C09108=1053.623,-71.148,432.234,170.544,29.693,155.607
C09109=1053.617,-71.397,432.246,170.542,29.692,155.607
C09110=1053.611,-71.647,432.257,170.540,29.691,155.607
C09111=1053.606,-71.896,432.269,170.538,29.689,155.606
C09112=1053.599,-72.147,432.280,170.536,29.688,155.606
C09113=1053.593,-72.396,432.292,170.535,29.686,155.606
C09114=1053.587,-72.646,432.303,170.533,29.685,155.606
C09115=1053.582,-72.895,432.315,170.531,29.684,155.606
C09116=1053.575,-73.145,432.327,170.529,29.683,155.606
C09117=1053.569,-73.394,432.338,170.527,29.681,155.606
C09118=1053.563,-73.644,432.349,170.524,29.679,155.606
C09119=1053.556,-73.894,432.361,170.523,29.679,155.606
C09120=1053.551,-74.144,432.373,170.521,29.677,155.606
C09121=1053.545,-74.394,432.384,170.519,29.676,155.606
C09122=1053.538,-74.643,432.394,170.517,29.675,155.605
C09123=1053.532,-74.892,432.406,170.515,29.673,155.605
C09124=1053.526,-75.142,432.417,170.513,29.672,155.605
C09125=1053.519,-75.392,432.429,170.511,29.671,155.605
C09126=1053.514,-75.641,432.440,170.510,29.670,155.605
C09127=1053.507,-75.891,432.451,170.508,29.669,155.605
C09128=1053.501,-76.141,432.462,170.505,29.668,155.605
C09129=1053.495,-76.390,432.474,170.503,29.666,155.605
C09130=1053.489,-76.640,432.485,170.501,29.665,155.605
C09131=1053.483,-76.890,432.496,170.499,29.663,155.605
C09132=1053.476,-77.140,432.508,170.498,29.662,155.605
C09133=1053.470,-77.389,432.519,170.496,29.661,155.605
C09134=1053.464,-77.639,432.530,170.494,29.660,155.604
C09135=1053.458,-77.889,432.541,170.492,29.659,155.604
C09136=1053.452,-78.138,432.553,170.490,29.658,155.604
C09137=1053.446,-78.388,432.564,170.487,29.657,155.604
C09138=1053.440,-78.638,432.575,170.486,29.655,155.604
C09139=1053.434,-78.887,432.586,170.484,29.654,155.604
C09140=1053.427,-79.137,432.598,170.482,29.653,155.604
C09141=1053.421,-79.386,432.609,170.480,29.651,155.604
C09142=1053.415,-79.637,432.620,170.478,29.651,155.604
C09143=1053.409,-79.886,432.631,170.476,29.650,155.604
C09144=1053.402,-80.136,432.642,170.474,29.649,155.604
C09145=1053.396,-80.385,432.653,170.473,29.647,155.604
C09146=1053.390,-80.635,432.665,170.470,29.646,155.604
C09147=1053.384,-80.885,432.675,170.468,29.645,155.604
C09148=1053.377,-81.134,432.686,170.466,29.644,155.604
C09149=1053.371,-81.384,432.697,170.464,29.643,155.604
C09150=1053.365,-81.634,432.708,170.462,29.642,155.604
C09151=1053.359,-81.884,432.719,170.460,29.641,155.604
C09152=1053.352,-82.134,432.730,170.459,29.640,155.604
C09153=1053.346,-82.382,432.741,170.457,29.638,155.603
C09154=1053.339,-82.666,432.754,170.454,29.637,155.603
C09155=1053.332,-82.949,432.766,170.452,29.636,155.603
C09156=1053.325,-83.233,432.778,170.449,29.635,155.603
C09157=1053.318,-83.517,432.791,170.447,29.633,155.603
C09158=1053.312,-83.767,432.802,170.446,29.632,155.603
C09159=1053.305,-84.017,432.812,170.444,29.631,155.603
C09160=1053.299,-84.266,432.823,170.441,29.630,155.603
C09161=1053.293,-84.516,432.835,170.439,29.629,155.603
C09162=1053.286,-84.766,432.845,170.437,29.628,155.603
C09163=1053.281,-85.015,432.856,170.435,29.627,155.603
C09164=1053.274,-85.265,432.867,170.433,29.626,155.603
C09165=1053.268,-85.515,432.877,170.431,29.625,155.603
C09166=1053.262,-85.765,432.889,170.430,29.624,155.603
C09167=1053.256,-86.014,432.899,170.428,29.623,155.603
C09168=1053.250,-86.264,432.910,170.425,29.622,155.603
C09169=1053.243,-86.514,432.921,170.423,29.621,155.603
C09170=1053.237,-86.763,432.932,170.421,29.620,155.603
C09171=1053.231,-87.013,432.943,170.419,29.619,155.603
C09172=1053.224,-87.262,432.953,170.417,29.618,155.603
C09173=1053.219,-87.512,432.964,170.416,29.617,155.603
C09174=1053.212,-87.762,432.975,170.414,29.616,155.603
C09175=1053.206,-88.011,432.986,170.411,29.615,155.603
C09176=1053.200,-88.261,432.997,170.409,29.614,155.603
C09177=1053.194,-88.512,433.007,170.407,29.613,155.602
C09178=1053.188,-88.761,433.017,170.405,29.612,155.602
C09179=1053.182,-89.010,433.028,170.403,29.611,155.602
C09180=1053.176,-89.260,433.040,170.402,29.610,155.602
C09181=1053.169,-89.510,433.050,170.400,29.609,155.602
C09182=1053.163,-89.759,433.061,170.397,29.608,155.602
C09183=1053.156,-90.009,433.071,170.395,29.607,155.602
C09184=1053.151,-90.258,433.082,170.393,29.606,155.602
C09185=1053.145,-90.509,433.092,170.391,29.605,155.602
C09186=1053.138,-90.758,433.103,170.389,29.604,155.602
C09187=1053.132,-91.008,433.114,170.388,29.603,155.602
C09188=1053.127,-91.257,433.125,170.386,29.602,155.602
C09189=1053.119,-91.507,433.135,170.384,29.601,155.602
C09190=1053.114,-91.757,433.146,170.381,29.600,155.602
C09191=1053.108,-92.007,433.156,170.379,29.599,155.602
C09192=1053.102,-92.256,433.167,170.377,29.598,155.602
C09193=1053.095,-92.506,433.178,170.375,29.597,155.602
C09194=1053.089,-92.755,433.188,170.374,29.596,155.602
C09195=1053.084,-93.006,433.198,170.372,29.595,155.602
C09196=1053.078,-93.255,433.209,170.370,29.594,155.602
C09197=1053.071,-93.505,433.220,170.367,29.593,155.602
C09198=1053.065,-93.754,433.231,170.365,29.592,155.602
C09199=1053.059,-94.004,433.240,170.363,29.591,155.602
C09200=1053.053,-94.254,433.251,170.361,29.590,155.602
C09201=1053.047,-94.504,433.263,170.359,29.589,155.602
C09202=1053.041,-94.754,433.272,170.358,29.588,155.602
C09203=1053.035,-95.003,433.283,170.355,29.587,155.602
C09204=1053.028,-95.252,433.293,170.353,29.586,155.602
C09205=1053.023,-95.503,433.303,170.351,29.586,155.602
C09206=1053.017,-95.753,433.315,170.349,29.585,155.602
C09207=1053.010,-96.002,433.325,170.347,29.584,155.602
C09208=1053.004,-96.251,433.336,170.345,29.583,155.602
C09209=1052.998,-96.501,433.345,170.344,29.582,155.602
C09210=1052.992,-96.751,433.356,170.341,29.580,155.602
C09211=1052.986,-97.001,433.367,170.339,29.579,155.602
C09212=1052.980,-97.251,433.377,170.337,29.579,155.602
C09213=1052.974,-97.500,433.388,170.335,29.578,155.602
C09214=1052.968,-97.750,433.398,170.333,29.577,155.602
C09215=1052.962,-97.999,433.408,170.331,29.576,155.602
C09216=1052.956,-98.250,433.418,170.329,29.576,155.602
C09217=1052.949,-98.499,433.429,170.327,29.574,155.602
C09218=1052.942,-98.785,433.440,170.325,29.573,155.602
C09219=1052.935,-99.071,433.452,170.322,29.573,155.602
C09220=1052.928,-99.357,433.463,170.320,29.572,155.602
C09221=1052.921,-99.643,433.475,170.317,29.571,155.602
C09222=1052.915,-99.893,433.486,170.315,29.570,155.602
C09223=1052.909,-100.142,433.496,170.313,29.569,155.602
C09224=1052.902,-100.392,433.506,170.311,29.568,155.602
C09225=1052.896,-100.642,433.517,170.310,29.568,155.602
C09226=1052.890,-100.891,433.527,170.308,29.567,155.602
C09227=1052.884,-101.141,433.537,170.305,29.566,155.602
C09228=1052.878,-101.391,433.547,170.303,29.565,155.602
C09229=1052.872,-101.641,433.557,170.301,29.564,155.602
C09230=1052.865,-101.890,433.567,170.299,29.564,155.602
C09231=1052.860,-102.141,433.577,170.297,29.563,155.602
C09232=1052.853,-102.390,433.588,170.295,29.562,155.602
C09233=1052.847,-102.640,433.597,170.293,29.561,155.602
C09234=1052.841,-102.889,433.608,170.291,29.560,155.602
C09235=1052.835,-103.139,433.618,170.289,29.560,155.602
C09236=1052.828,-103.388,433.628,170.287,29.559,155.602
C09237=1052.823,-103.638,433.638,170.285,29.559,155.602
C09238=1052.817,-103.888,433.648,170.283,29.558,155.602
C09239=1052.810,-104.138,433.658,170.280,29.556,155.602
C09240=1052.804,-104.388,433.668,170.278,29.556,155.602
C09241=1052.798,-104.638,433.678,170.276,29.555,155.602
C09242=1052.792,-104.887,433.688,170.275,29.555,155.602
C09243=1052.786,-105.137,433.698,170.273,29.554,155.602
C09244=1052.780,-105.386,433.709,170.271,29.553,155.602
C09245=1052.774,-105.636,433.718,170.268,29.552,155.602
C09246=1052.767,-105.886,433.728,170.266,29.552,155.602
C09247=1052.761,-106.135,433.738,170.264,29.551,155.602
C09248=1052.756,-106.385,433.748,170.262,29.550,155.602
C09249=1052.749,-106.635,433.758,170.260,29.549,155.602
C09250=1052.743,-106.885,433.767,170.258,29.549,155.602
C09251=1052.737,-107.134,433.778,170.256,29.548,155.602
C09252=1052.731,-107.384,433.788,170.254,29.547,155.602
C09253=1052.725,-107.634,433.798,170.252,29.547,155.602
C09254=1052.718,-107.884,433.808,170.250,29.546,155.602
C09255=1052.712,-108.133,433.818,170.248,29.546,155.602
C09256=1052.706,-108.383,433.827,170.245,29.544,155.602
C09257=1052.700,-108.633,433.837,170.243,29.544,155.603
C09258=1052.693,-108.883,433.846,170.241,29.544,155.603
C09259=1052.687,-109.132,433.857,170.239,29.543,155.603
C09260=1052.681,-109.382,433.867,170.237,29.542,155.603
C09261=1052.675,-109.632,433.876,170.236,29.542,155.603
C09262=1052.669,-109.882,433.886,170.233,29.541,155.603
C09263=1052.663,-110.131,433.896,170.231,29.540,155.603
C09264=1052.656,-110.381,433.906,170.229,29.540,155.603
C09265=1052.650,-110.630,433.915,170.227,29.539,155.603
C09266=1052.644,-110.880,433.925,170.225,29.539,155.603
C09267=1052.638,-111.130,433.935,170.222,29.538,155.603
C09268=1052.632,-111.380,433.944,170.220,29.538,155.603
C09269=1052.626,-111.630,433.954,170.218,29.537,155.603
C09270=1052.620,-111.879,433.965,170.217,29.536,155.603
C09271=1052.614,-112.129,433.974,170.215,29.536,155.603
C09272=1052.607,-112.379,433.984,170.213,29.535,155.603
C09273=1052.601,-112.629,433.993,170.210,29.534,155.603
C09274=1052.595,-112.878,434.003,170.208,29.534,155.603
C09275=1052.589,-113.128,434.012,170.206,29.534,155.603
C09276=1052.583,-113.378,434.022,170.204,29.533,155.603
C09277=1052.577,-113.628,434.032,170.202,29.532,155.603
C09278=1052.570,-113.878,434.041,170.199,29.532,155.604
C09279=1052.564,-114.127,434.051,170.197,29.531,155.604
C09280=1052.558,-114.377,434.060,170.196,29.530,155.604
C09281=1052.552,-114.626,434.070,170.194,29.530,155.604
C09282=1052.545,-114.911,434.081,170.191,29.529,155.604
C09283=1052.538,-115.194,434.092,170.189,29.529,155.604
C09284=1052.531,-115.478,434.103,170.186,29.528,155.604
C09285=1052.524,-115.763,434.113,170.184,29.527,155.604
C09286=1052.518,-116.013,434.123,170.182,29.527,155.604
C09287=1052.512,-116.262,434.132,170.180,29.527,155.604
C09288=1052.506,-116.511,434.142,170.177,29.526,155.604
C09289=1052.500,-116.761,434.151,170.175,29.526,155.604
C09290=1052.494,-117.011,434.161,170.173,29.525,155.604
C09291=1052.488,-117.261,434.170,170.172,29.525,155.604
C09292=1052.482,-117.511,434.180,170.170,29.524,155.605
C09293=1052.475,-117.760,434.189,170.167,29.523,155.605
C09294=1052.469,-118.010,434.199,170.165,29.523,155.605
C09295=1052.463,-118.260,434.209,170.163,29.522,155.605
C09296=1052.457,-118.510,434.218,170.161,29.522,155.605
C09297=1052.450,-118.759,434.227,170.159,29.522,155.605
C09298=1052.444,-119.008,434.236,170.156,29.521,155.605
C09299=1052.438,-119.258,434.246,170.154,29.521,155.605
C09300=1052.432,-119.509,434.255,170.152,29.520,155.605
C09301=1052.426,-119.758,434.264,170.150,29.520,155.605
C09302=1052.420,-120.008,434.274,170.149,29.520,155.605
C09303=1052.414,-120.258,434.283,170.146,29.519,155.605
C09304=1052.408,-120.508,434.293,170.144,29.519,155.605
C09305=1052.402,-120.757,434.302,170.142,29.518,155.606
C09306=1052.395,-121.006,434.311,170.140,29.518,155.606
C09307=1052.389,-121.257,434.320,170.138,29.518,155.606
C09308=1052.383,-121.507,434.330,170.135,29.517,155.606
C09309=1052.377,-121.756,434.339,170.133,29.517,155.606
C09310=1052.371,-122.006,434.349,170.131,29.516,155.606
C09311=1052.365,-122.255,434.358,170.129,29.516,155.606
C09312=1052.359,-122.506,434.367,170.127,29.515,155.606
C09313=1052.352,-122.755,434.376,170.124,29.515,155.606
C09314=1052.346,-123.005,434.385,170.123,29.514,155.606
C09315=1052.340,-123.255,434.395,170.121,29.514,155.606
C09316=1052.335,-123.504,434.404,170.119,29.514,155.606
C09317=1052.329,-123.754,434.413,170.117,29.513,155.607
C09318=1052.322,-124.005,434.423,170.114,29.513,155.607
C09319=1052.316,-124.255,434.432,170.112,29.513,155.607
C09320=1052.310,-124.506,434.441,170.110,29.513,155.607
C09321=1052.304,-124.755,434.450,170.108,29.512,155.607
C09322=1052.297,-125.006,434.458,170.106,29.512,155.607
C09323=1052.291,-125.255,434.468,170.103,29.511,155.607
C09324=1052.285,-125.505,434.478,170.101,29.511,155.607
C09325=1052.280,-125.755,434.486,170.099,29.510,155.607
C09326=1052.273,-126.004,434.495,170.097,29.511,155.608
C09327=1052.267,-126.254,434.505,170.095,29.510,155.608
C09328=1052.261,-126.505,434.513,170.093,29.510,155.608
C09329=1052.254,-126.754,434.522,170.091,29.509,155.608
C09330=1052.248,-127.003,434.532,170.089,29.509,155.608
C09331=1052.243,-127.254,434.540,170.087,29.509,155.608
C09332=1052.236,-127.503,434.549,170.085,29.509,155.608
C09333=1052.230,-127.752,434.559,170.082,29.508,155.608
C09334=1052.225,-128.003,434.568,170.080,29.508,155.608
C09335=1052.220,-128.252,434.578,170.078,29.507,155.608
C09336=1052.217,-128.502,434.589,170.076,29.505,155.608
C09337=1052.215,-128.752,434.600,170.075,29.503,155.608
C09338=1052.214,-129.004,434.612,170.074,29.500,155.607
C09339=1052.213,-129.254,434.625,170.072,29.498,155.607
C09340=1052.215,-129.504,434.638,170.071,29.494,155.607
C09341=1052.217,-129.754,434.652,170.070,29.490,155.606
C09342=1052.221,-130.005,434.667,170.069,29.485,155.605
C09343=1052.225,-130.255,434.682,170.068,29.480,155.604
C09344=1052.231,-130.507,434.698,170.068,29.475,155.603
C09345=1052.238,-130.757,434.715,170.067,29.468,155.602
C09346=1051.870,-130.779,434.495,170.020,29.636,155.635
C09347=1051.864,-130.530,434.479,170.021,29.643,155.636
C09348=1051.858,-130.280,434.463,170.021,29.648,155.637
C09349=1051.853,-130.028,434.447,170.023,29.653,155.638
C09350=1051.850,-129.778,434.433,170.023,29.658,155.638
C09351=1051.848,-129.527,434.419,170.025,29.662,155.639
C09352=1051.847,-129.277,434.406,170.025,29.666,155.640
C09353=1051.846,-129.026,434.393,170.027,29.669,155.640
C09354=1051.847,-128.776,434.380,170.029,29.671,155.640
C09355=1051.849,-128.526,434.369,170.030,29.674,155.641
C09356=1051.852,-128.276,434.358,170.032,29.675,155.641
C09357=1051.857,-128.025,434.348,170.034,29.676,155.641
C09358=1051.862,-127.776,434.339,170.036,29.677,155.641
C09359=1051.868,-127.526,434.329,170.038,29.677,155.641
C09360=1051.874,-127.277,434.321,170.040,29.677,155.641
C09361=1051.881,-127.027,434.312,170.042,29.678,155.641
C09362=1051.887,-126.777,434.302,170.045,29.678,155.640
C09363=1051.893,-126.527,434.294,170.047,29.678,155.640
C09364=1051.899,-126.278,434.285,170.049,29.678,155.640
C09365=1051.905,-126.028,434.275,170.050,29.679,155.640
C09366=1051.911,-125.778,434.267,170.052,29.679,155.640
C09367=1051.918,-125.528,434.258,170.055,29.680,155.640
C09368=1051.924,-125.279,434.248,170.057,29.680,155.640
C09369=1051.929,-125.029,434.240,170.059,29.680,155.640
C09370=1051.935,-124.779,434.230,170.061,29.680,155.640
C09371=1051.942,-124.530,434.221,170.064,29.681,155.639
C09372=1051.948,-124.279,434.212,170.066,29.681,155.639
C09373=1051.954,-124.029,434.203,170.068,29.682,155.639
C09374=1051.960,-123.780,434.193,170.070,29.682,155.639
C09375=1051.966,-123.531,434.184,170.072,29.682,155.639
C09376=1051.973,-123.280,434.176,170.075,29.683,155.639
C09377=1051.979,-123.031,434.166,170.077,29.683,155.639
C09378=1051.985,-122.781,434.156,170.079,29.683,155.639
C09379=1051.991,-122.532,434.147,170.080,29.683,155.639
C09380=1051.996,-122.281,434.138,170.082,29.684,155.639
C09381=1052.003,-122.032,434.129,170.085,29.684,155.639
C09382=1052.010,-121.782,434.120,170.087,29.685,155.638
C09383=1052.016,-121.532,434.110,170.089,29.685,155.638
C09384=1052.021,-121.283,434.101,170.091,29.685,155.638
C09385=1052.027,-121.033,434.092,170.093,29.686,155.638
C09386=1052.033,-120.783,434.083,170.096,29.686,155.638
C09387=1052.040,-120.533,434.073,170.098,29.687,155.638
C09388=1052.046,-120.283,434.064,170.100,29.687,155.638
C09389=1052.053,-120.034,434.055,170.102,29.687,155.638
C09390=1052.059,-119.784,434.045,170.104,29.688,155.638
C09391=1052.064,-119.535,434.036,170.106,29.688,155.638
C09392=1052.070,-119.285,434.027,170.108,29.689,155.638
C09393=1052.076,-119.035,434.017,170.110,29.689,155.638
C09394=1052.083,-118.785,434.008,170.112,29.690,155.637
C09395=1052.089,-118.535,433.998,170.114,29.690,155.637
C09396=1052.095,-118.285,433.989,170.117,29.690,155.637
C09397=1052.101,-118.036,433.979,170.119,29.691,155.637
C09398=1052.107,-117.786,433.970,170.121,29.692,155.637
C09399=1052.113,-117.537,433.960,170.123,29.692,155.637
C09400=1052.120,-117.287,433.951,170.125,29.693,155.637
C09401=1052.126,-117.037,433.942,170.128,29.693,155.637
C09402=1052.132,-116.788,433.932,170.130,29.694,155.637
C09403=1052.138,-116.538,433.923,170.131,29.694,155.637
C09404=1052.144,-116.288,433.913,170.133,29.694,155.637
C09405=1052.151,-116.038,433.904,170.135,29.695,155.637
C09406=1052.157,-115.788,433.894,170.138,29.695,155.637
C09407=1052.164,-115.503,433.883,170.140,29.696,155.637
C09408=1052.170,-115.219,433.872,170.143,29.697,155.636
C09409=1052.177,-114.935,433.861,170.145,29.697,155.636
C09410=1052.184,-114.650,433.851,170.148,29.698,155.636
C09411=1052.191,-114.400,433.841,170.150,29.698,155.636
C09412=1052.197,-114.150,433.831,170.152,29.698,155.636
C09413=1052.203,-113.900,433.822,170.153,29.699,155.636
C09414=1052.209,-113.650,433.812,170.155,29.700,155.636
C09415=1052.215,-113.401,433.803,170.158,29.700,155.636
C09416=1052.221,-113.151,433.793,170.160,29.701,155.636
C09417=1052.228,-112.901,433.784,170.162,29.702,155.636
C09418=1052.234,-112.651,433.774,170.164,29.702,155.636
C09419=1052.240,-112.401,433.764,170.166,29.702,155.636
C09420=1052.246,-112.152,433.754,170.169,29.704,155.636
C09421=1052.252,-111.902,433.744,170.171,29.704,155.636
C09422=1052.258,-111.652,433.734,170.173,29.704,155.636
C09423=1052.264,-111.403,433.725,170.175,29.705,155.636
C09424=1052.270,-111.153,433.715,170.176,29.706,155.636
C09425=1052.276,-110.903,433.706,170.178,29.706,155.636
C09426=1052.283,-110.653,433.696,170.181,29.707,155.635
C09427=1052.289,-110.404,433.686,170.183,29.708,155.635
C09428=1052.295,-110.154,433.676,170.185,29.708,155.635
C09429=1052.301,-109.904,433.667,170.187,29.708,155.635
C09430=1052.307,-109.654,433.657,170.189,29.709,155.635
C09431=1052.313,-109.404,433.647,170.192,29.710,155.635
C09432=1052.320,-109.155,433.637,170.194,29.710,155.635
C09433=1052.326,-108.906,433.627,170.196,29.711,155.635
C09434=1052.332,-108.656,433.618,170.197,29.712,155.635
C09435=1052.338,-108.406,433.608,170.199,29.712,155.635
C09436=1052.345,-108.157,433.598,170.202,29.713,155.635
C09437=1052.351,-107.907,433.588,170.204,29.714,155.635
C09438=1052.356,-107.657,433.578,170.206,29.714,155.635
C09439=1052.362,-107.407,433.568,170.208,29.715,155.635
C09440=1052.369,-107.158,433.558,170.210,29.715,155.635
C09441=1052.375,-106.908,433.549,170.212,29.716,155.635
C09442=1052.381,-106.658,433.539,170.215,29.717,155.635
C09443=1052.387,-106.408,433.529,170.217,29.717,155.635
C09444=1052.393,-106.159,433.519,170.218,29.718,155.635
C09445=1052.399,-105.909,433.509,170.220,29.719,155.635
C09446=1052.405,-105.659,433.499,170.222,29.720,155.635
C09447=1052.412,-105.409,433.488,170.225,29.720,155.635
C09448=1052.418,-105.159,433.479,170.227,29.721,155.635
C09449=1052.424,-104.910,433.469,170.229,29.722,155.635
C09450=1052.431,-104.660,433.459,170.231,29.723,155.635
C09451=1052.436,-104.410,433.449,170.233,29.723,155.635
C09452=1052.442,-104.161,433.438,170.235,29.724,155.635
C09453=1052.449,-103.911,433.429,170.237,29.724,155.634
C09454=1052.454,-103.661,433.419,170.239,29.725,155.635
C09455=1052.461,-103.412,433.408,170.241,29.726,155.635
C09456=1052.467,-103.162,433.399,170.243,29.727,155.634
C09457=1052.473,-102.912,433.387,170.245,29.728,155.635
C09458=1052.479,-102.662,433.378,170.247,29.728,155.634
C09459=1052.485,-102.412,433.368,170.250,29.729,155.634
C09460=1052.491,-102.163,433.357,170.252,29.730,155.634
C09461=1052.497,-101.913,433.348,170.254,29.731,155.634
C09462=1052.504,-101.664,433.338,170.255,29.732,155.634
C09463=1052.511,-101.341,433.325,170.258,29.732,155.634
C09464=1052.520,-101.019,433.312,170.261,29.733,155.634
C09465=1052.528,-100.697,433.298,170.264,29.735,155.634
C09466=1052.536,-100.375,433.285,170.266,29.736,155.634
C09467=1052.541,-100.144,433.276,170.268,29.736,155.634
C09468=1052.547,-99.912,433.266,170.270,29.737,155.634
C09469=1052.553,-99.680,433.257,170.272,29.737,155.634
C09470=1052.558,-99.448,433.247,170.273,29.738,155.634
C09471=1052.565,-99.217,433.237,170.275,29.739,155.634
C09472=1052.570,-98.986,433.228,170.277,29.740,155.634
C09473=1052.575,-98.754,433.218,170.279,29.741,155.634
C09474=1052.581,-98.522,433.209,170.281,29.741,155.634
C09475=1052.588,-98.273,433.199,170.284,29.742,155.634
C09476=1052.593,-98.023,433.189,170.286,29.743,155.634
C09477=1052.600,-97.773,433.178,170.288,29.744,155.634
C09478=1052.606,-97.523,433.167,170.290,29.745,155.634
C09479=1052.612,-97.273,433.158,170.291,29.746,155.634
C09480=1052.618,-97.024,433.147,170.293,29.746,155.634
C09481=1052.624,-96.774,433.137,170.296,29.747,155.634
C09482=1052.631,-96.524,433.126,170.298,29.748,155.634
C09483=1052.637,-96.275,433.116,170.300,29.749,155.634
C09484=1052.643,-96.025,433.106,170.302,29.750,155.634
C09485=1052.648,-95.775,433.095,170.304,29.751,155.634
C09486=1052.655,-95.526,433.085,170.306,29.752,155.634
C09487=1052.661,-95.275,433.074,170.308,29.753,155.634
C09488=1052.667,-95.026,433.064,170.310,29.754,155.634
C09489=1052.673,-94.776,433.053,170.312,29.755,155.634
C09490=1052.678,-94.526,433.043,170.314,29.755,155.634
C09491=1052.685,-94.277,433.032,170.316,29.756,155.634
C09492=1052.691,-94.027,433.021,170.318,29.757,155.634
C09493=1052.698,-93.778,433.011,170.320,29.758,155.635
C09494=1052.703,-93.528,433.001,170.322,29.760,155.635
C09495=1052.709,-93.278,432.990,170.324,29.760,155.634
C09496=1052.716,-93.028,432.979,170.326,29.761,155.634
C09497=1052.722,-92.779,432.968,170.328,29.762,155.635
C09498=1052.728,-92.529,432.959,170.330,29.763,155.635
C09499=1052.734,-92.280,432.948,170.332,29.764,155.635
C09500=1052.740,-92.029,432.937,170.334,29.765,155.635
C09501=1052.746,-91.780,432.926,170.337,29.766,155.635
C09502=1052.752,-91.530,432.916,170.338,29.767,155.635
C09503=1052.758,-91.281,432.905,170.340,29.768,155.635
C09504=1052.765,-91.031,432.895,170.342,29.769,155.635
C09505=1052.770,-90.781,432.884,170.344,29.770,155.635
C09506=1052.777,-90.532,432.874,170.346,29.771,155.635
C09507=1052.783,-90.282,432.862,170.348,29.772,155.635
C09508=1052.789,-90.032,432.852,170.351,29.773,155.635
C09509=1052.795,-89.783,432.842,170.353,29.774,155.635
C09510=1052.802,-89.532,432.831,170.354,29.775,155.635
C09511=1052.807,-89.283,432.820,170.356,29.775,155.635
C09512=1052.814,-89.034,432.809,170.358,29.776,155.635
C09513=1052.820,-88.783,432.798,170.360,29.777,155.635
C09514=1052.826,-88.534,432.787,170.362,29.778,155.635
C09515=1052.832,-88.285,432.777,170.365,29.780,155.635
C09516=1052.839,-88.035,432.766,170.367,29.781,155.635
C09517=1052.844,-87.785,432.756,170.368,29.782,155.635
C09518=1052.851,-87.535,432.745,170.370,29.783,155.635
C09519=1052.857,-87.285,432.734,170.372,29.784,155.635
C09520=1052.863,-87.036,432.723,170.374,29.785,155.635
C09521=1052.870,-86.786,432.713,170.376,29.786,155.635
C09522=1052.875,-86.536,432.702,170.379,29.787,155.635
C09523=1052.881,-86.287,432.691,170.381,29.788,155.635
C09524=1052.888,-86.037,432.680,170.383,29.789,155.635
C09525=1052.894,-85.787,432.669,170.384,29.790,155.635
C09526=1052.900,-85.538,432.658,170.386,29.791,155.635
C09527=1052.907,-85.288,432.648,170.388,29.792,155.636
C09528=1052.913,-85.039,432.637,170.390,29.793,155.636
C09529=1052.919,-84.788,432.626,170.393,29.794,155.636
C09530=1052.925,-84.539,432.615,170.395,29.795,155.636
C09531=1052.932,-84.289,432.604,170.397,29.796,155.636
C09532=1052.937,-84.040,432.593,170.398,29.797,155.636
C09533=1052.943,-83.790,432.582,170.400,29.798,155.636
C09534=1052.950,-83.540,432.572,170.402,29.799,155.636
C09535=1052.957,-83.256,432.559,170.405,29.800,155.636
C09536=1052.964,-82.973,432.547,170.407,29.801,155.636
C09537=1052.971,-82.689,432.534,170.410,29.803,155.636
C09538=1052.979,-82.405,432.522,170.412,29.804,155.636
C09539=1052.985,-82.156,432.510,170.413,29.805,155.636
C09540=1052.991,-81.906,432.499,170.415,29.806,155.636
C09541=1052.997,-81.657,432.489,170.417,29.807,155.636
C09542=1053.004,-81.407,432.478,170.419,29.808,155.636
C09543=1053.009,-81.157,432.467,170.422,29.809,155.636
C09544=1053.016,-80.907,432.456,170.424,29.811,155.636
C09545=1053.022,-80.658,432.445,170.426,29.812,155.636
C09546=1053.029,-80.408,432.434,170.427,29.813,155.636
C09547=1053.035,-80.159,432.422,170.429,29.814,155.636
C09548=1053.041,-79.909,432.411,170.431,29.815,155.636
C09549=1053.048,-79.659,432.401,170.433,29.816,155.637
C09550=1053.054,-79.409,432.390,170.435,29.817,155.637
C09551=1053.060,-79.160,432.379,170.438,29.819,155.637
C09552=1053.066,-78.910,432.367,170.440,29.820,155.637
C09553=1053.072,-78.661,432.356,170.441,29.820,155.637
C09554=1053.078,-78.410,432.345,170.443,29.822,155.637
C09555=1053.084,-78.161,432.334,170.445,29.823,155.637
C09556=1053.091,-77.911,432.322,170.447,29.824,155.637
C09557=1053.096,-77.662,432.311,170.449,29.826,155.637
C09558=1053.103,-77.412,432.300,170.451,29.827,155.637
C09559=1053.109,-77.162,432.289,170.453,29.828,155.637
C09560=1053.115,-76.913,432.277,170.455,29.829,155.637
C09561=1053.121,-76.663,432.266,170.457,29.830,155.637
C09562=1053.127,-76.413,432.255,170.459,29.831,155.637
C09563=1053.133,-76.164,432.243,170.461,29.833,155.638
C09564=1053.140,-75.914,432.232,170.463,29.834,155.638
C09565=1053.146,-75.664,432.221,170.465,29.835,155.638
C09566=1053.152,-75.415,432.209,170.466,29.836,155.638
C09567=1053.158,-75.165,432.198,170.468,29.837,155.638
C09568=1053.164,-74.915,432.187,170.470,29.838,155.638
C09569=1053.171,-74.666,432.175,170.473,29.840,155.638
C09570=1053.176,-74.416,432.164,170.475,29.841,155.638
C09571=1053.183,-74.166,432.153,170.477,29.842,155.638
C09572=1053.189,-73.917,432.141,170.479,29.844,155.638
C09573=1053.195,-73.667,432.130,170.480,29.845,155.638
C09574=1053.202,-73.417,432.119,170.482,29.846,155.638
C09575=1053.208,-73.168,432.107,170.484,29.847,155.638
C09576=1053.213,-72.917,432.095,170.486,29.849,155.639
C09577=1053.219,-72.668,432.084,170.488,29.850,155.639
C09578=1053.226,-72.418,432.073,170.490,29.851,155.639
C09579=1053.232,-72.169,432.061,170.491,29.853,155.639
C09580=1053.237,-71.919,432.049,170.494,29.854,155.639
C09581=1053.243,-71.670,432.038,170.496,29.856,155.639
C09582=1053.250,-71.420,432.026,170.498,29.857,155.639
C09583=1053.256,-71.171,432.015,170.500,29.858,155.639
C09584=1053.261,-70.920,432.003,170.502,29.859,155.639
C09585=1053.268,-70.671,431.991,170.503,29.861,155.640
C09586=1053.274,-70.421,431.980,170.505,29.863,155.640
C09587=1053.280,-70.172,431.968,170.507,29.864,155.640
C09588=1053.285,-69.922,431.957,170.509,29.865,155.640
C09589=1053.292,-69.672,431.945,170.511,29.866,155.640
C09590=1053.298,-69.423,431.934,170.513,29.868,155.640
C09591=1053.304,-69.173,431.922,170.515,29.869,155.640
C09592=1053.310,-68.923,431.910,170.516,29.870,155.640
C09593=1053.316,-68.674,431.898,170.519,29.872,155.640
C09594=1053.323,-68.424,431.886,170.521,29.873,155.640
C09595=1053.329,-68.174,431.875,170.523,29.875,155.641
C09596=1053.334,-67.925,431.863,170.525,29.876,155.641
C09597=1053.341,-67.675,431.852,170.527,29.877,155.641
C09598=1053.347,-67.426,431.840,170.528,29.879,155.641
C09599=1053.354,-67.144,431.826,170.530,29.880,155.641
C09600=1053.361,-66.863,431.814,170.533,29.881,155.641
C09601=1053.368,-66.581,431.800,170.535,29.883,155.641
C09602=1053.374,-66.300,431.787,170.537,29.885,155.641
C09603=1053.381,-66.049,431.775,170.538,29.886,155.642
C09604=1053.387,-65.800,431.764,170.540,29.887,155.642
C09605=1053.393,-65.551,431.751,170.543,29.889,155.642
C09606=1053.399,-65.300,431.740,170.545,29.891,155.642
C09607=1053.405,-65.052,431.728,170.547,29.892,155.642
C09608=1053.411,-64.802,431.716,170.549,29.893,155.642
C09609=1053.417,-64.551,431.705,170.550,29.895,155.642
C09610=1053.424,-64.302,431.693,170.552,29.896,155.642
C09611=1053.430,-64.053,431.681,170.554,29.897,155.642
C09612=1053.436,-63.803,431.669,170.556,29.899,155.643
C09613=1053.442,-63.553,431.657,170.558,29.900,155.643
C09614=1053.448,-63.304,431.646,170.560,29.901,155.643
C09615=1053.454,-63.054,431.633,170.562,29.903,155.643
C09616=1053.461,-62.805,431.621,170.563,29.905,155.643
C09617=1053.467,-62.554,431.610,170.565,29.906,155.643
C09618=1053.473,-62.305,431.598,170.567,29.907,155.643
C09619=1053.479,-62.056,431.586,170.569,29.909,155.643
C09620=1053.486,-61.806,431.574,170.572,29.910,155.643
C09621=1053.491,-61.556,431.562,170.574,29.911,155.644
C09622=1053.497,-61.307,431.550,170.575,29.913,155.644
C09623=1053.504,-61.057,431.538,170.577,29.915,155.644
C09624=1053.510,-60.807,431.526,170.579,29.916,155.644
C09625=1053.517,-60.558,431.514,170.581,29.917,155.644
C09626=1053.523,-60.308,431.502,170.583,29.919,155.644
C09627=1053.528,-60.058,431.490,170.585,29.920,155.644
C09628=1053.535,-59.809,431.479,170.586,29.921,155.644
C09629=1053.542,-59.559,431.467,170.588,29.923,155.645
C09630=1053.548,-59.309,431.454,170.590,29.925,155.645
C09631=1053.554,-59.060,431.442,170.592,29.925,155.645
C09632=1053.559,-58.811,431.430,170.594,29.927,155.645
C09633=1053.566,-58.561,431.418,170.596,29.929,155.645
C09634=1053.572,-58.311,431.407,170.597,29.930,155.645
C09635=1053.578,-58.061,431.394,170.599,29.932,155.645
C09636=1053.585,-57.811,431.382,170.601,29.933,155.645
C09637=1053.592,-57.562,431.370,170.603,29.934,155.646
C09638=1053.597,-57.313,431.358,170.606,29.936,155.646
C09639=1053.604,-57.063,431.346,170.608,29.938,155.646
C09640=1053.610,-56.813,431.334,170.609,29.939,155.646
C09641=1053.616,-56.564,431.322,170.611,29.940,155.646
C09642=1053.623,-56.314,431.310,170.613,29.942,155.646
C09643=1053.629,-56.064,431.297,170.615,29.943,155.646
C09644=1053.635,-55.815,431.285,170.617,29.945,155.647
C09645=1053.642,-55.565,431.273,170.619,29.946,155.647
C09646=1053.647,-55.316,431.261,170.620,29.948,155.647
C09647=1053.654,-55.066,431.249,170.622,29.949,155.647
C09648=1053.660,-54.816,431.236,170.624,29.951,155.647
C09649=1053.667,-54.567,431.224,170.626,29.952,155.647
C09650=1053.673,-54.317,431.212,170.628,29.953,155.647
C09651=1053.679,-54.067,431.200,170.630,29.955,155.647
C09652=1053.686,-53.818,431.188,170.631,29.956,155.648
C09653=1053.692,-53.568,431.175,170.633,29.958,155.648
C09654=1053.698,-53.318,431.163,170.635,29.960,155.648
C09655=1053.705,-53.069,431.151,170.637,29.961,155.648
C09656=1053.711,-52.819,431.139,170.639,29.962,155.648
C09657=1053.717,-52.569,431.127,170.641,29.964,155.648
C09658=1053.723,-52.319,431.114,170.642,29.965,155.648
C09659=1053.730,-52.071,431.102,170.644,29.967,155.649
C09660=1053.736,-51.821,431.090,170.647,29.969,155.649
C09661=1053.742,-51.572,431.078,170.649,29.970,155.649
C09662=1053.749,-51.322,431.066,170.651,29.971,155.649
C09663=1053.756,-51.041,431.052,170.652,29.973,155.649
C09664=1053.763,-50.761,431.038,170.654,29.975,155.649
C09665=1053.770,-50.481,431.023,170.656,29.977,155.650
C09666=1053.778,-50.200,431.010,170.659,29.978,155.650
C09667=1053.783,-49.951,430.998,170.661,29.980,155.650
C09668=1053.789,-49.701,430.985,170.663,29.981,155.650
C09669=1053.795,-49.452,430.973,170.664,29.983,155.650
C09670=1053.802,-49.203,430.960,170.666,29.985,155.650
C09671=1053.808,-48.953,430.947,170.668,29.986,155.650
C09672=1053.814,-48.703,430.935,170.670,29.988,155.651
C09673=1053.820,-48.453,430.922,170.672,29.989,155.651
C09674=1053.827,-48.204,430.910,170.673,29.992,155.651
C09675=1053.832,-47.954,430.897,170.675,29.993,155.651
C09676=1053.838,-47.704,430.884,170.677,29.995,155.651
C09677=1053.844,-47.454,430.872,170.679,29.996,155.651
C09678=1053.851,-47.205,430.859,170.681,29.998,155.652
C09679=1053.857,-46.955,430.847,170.683,29.999,155.652
C09680=1053.863,-46.706,430.834,170.684,30.001,155.652
C09681=1053.869,-46.456,430.821,170.686,30.003,155.652
C09682=1053.876,-46.207,430.809,170.688,30.004,155.652
C09683=1053.882,-45.957,430.796,170.690,30.006,155.653
C09684=1053.888,-45.708,430.783,170.692,30.008,155.653
C09685=1053.894,-45.458,430.771,170.693,30.009,155.653
C09686=1053.901,-45.208,430.759,170.695,30.011,155.653
C09687=1053.907,-44.959,430.745,170.697,30.013,155.653
C09688=1053.913,-44.709,430.733,170.699,30.014,155.653
C09689=1053.919,-44.459,430.720,170.701,30.016,155.653
C09690=1053.925,-44.210,430.707,170.703,30.017,155.654
C09691=1053.931,-43.960,430.695,170.704,30.020,155.654
C09692=1053.937,-43.710,430.682,170.706,30.021,155.654
C09693=1053.944,-43.461,430.669,170.708,30.023,155.654
C09694=1053.949,-43.211,430.657,170.710,30.024,155.654
C09695=1053.956,-42.962,430.643,170.712,30.026,155.655
C09696=1053.962,-42.712,430.631,170.714,30.027,155.655
C09697=1053.969,-42.463,430.618,170.715,30.029,155.655
C09698=1053.974,-42.213,430.606,170.717,30.031,155.655
C09699=1053.980,-41.963,430.593,170.719,30.033,155.655
C09700=1053.987,-41.714,430.580,170.721,30.034,155.655
C09701=1053.993,-41.465,430.568,170.723,30.036,155.656
C09702=1053.999,-41.215,430.554,170.724,30.037,155.656
C09703=1054.005,-40.965,430.542,170.726,30.039,155.656
C09704=1054.012,-40.715,430.528,170.728,30.041,155.656
C09705=1054.018,-40.466,430.516,170.730,30.043,155.656
C09706=1054.024,-40.216,430.502,170.732,30.044,155.656
C09707=1054.031,-39.967,430.490,170.734,30.046,155.657
C09708=1054.037,-39.717,430.477,170.735,30.048,155.657
C09709=1054.043,-39.468,430.465,170.737,30.050,155.657
C09710=1054.049,-39.218,430.451,170.739,30.051,155.657
C09711=1054.055,-38.968,430.439,170.741,30.053,155.657
C09712=1054.062,-38.718,430.425,170.743,30.054,155.658
C09713=1054.069,-38.470,430.413,170.744,30.056,155.658
C09714=1054.074,-38.219,430.399,170.746,30.058,155.658
C09715=1054.080,-37.970,430.386,170.748,30.060,155.658
C09716=1054.086,-37.720,430.374,170.749,30.061,155.658
C09717=1054.092,-37.471,430.360,170.751,30.063,155.659
C09718=1054.099,-37.222,430.347,170.753,30.065,155.659
C09719=1054.105,-36.972,430.334,170.754,30.066,155.659
C09720=1054.111,-36.723,430.321,170.756,30.069,155.659
C09721=1054.117,-36.473,430.309,170.758,30.070,155.659
C09722=1054.123,-36.223,430.295,170.760,30.072,155.660
C09723=1054.130,-35.973,430.282,170.762,30.074,155.660
C09724=1054.136,-35.724,430.269,170.763,30.076,155.660
C09725=1054.142,-35.474,430.256,170.765,30.078,155.660
C09726=1054.148,-35.225,430.243,170.767,30.079,155.660
C09727=1054.155,-34.945,430.228,170.769,30.081,155.661
C09728=1054.162,-34.665,430.213,170.771,30.083,155.661
C09729=1054.169,-34.385,430.199,170.773,30.085,155.661
C09730=1054.176,-34.105,430.184,170.775,30.088,155.661
C09731=1054.182,-33.856,430.171,170.777,30.089,155.661
C09732=1054.188,-33.607,430.157,170.779,30.091,155.662
C09733=1054.194,-33.357,430.145,170.781,30.093,155.662
C09734=1054.201,-33.107,430.131,170.782,30.094,155.662
C09735=1054.206,-32.857,430.117,170.784,30.096,155.662
C09736=1054.213,-32.608,430.104,170.786,30.098,155.662
C09737=1054.218,-32.358,430.091,170.788,30.100,155.663
C09738=1054.225,-32.109,430.078,170.790,30.102,155.663
C09739=1054.231,-31.859,430.065,170.791,30.103,155.663
C09740=1054.238,-31.610,430.051,170.792,30.105,155.663
C09741=1054.244,-31.361,430.038,170.794,30.107,155.664
C09742=1054.250,-31.111,430.025,170.796,30.109,155.664
C09743=1054.257,-30.861,430.012,170.798,30.111,155.664
C09744=1054.263,-30.611,429.999,170.800,30.112,155.664
C09745=1054.268,-30.362,429.985,170.801,30.114,155.664
C09746=1054.275,-30.113,429.971,170.803,30.116,155.665
C09747=1054.281,-29.863,429.958,170.805,30.118,155.665
C09748=1054.287,-29.613,429.945,170.807,30.120,155.665
C09749=1054.293,-29.363,429.932,170.809,30.121,155.665
C09750=1054.300,-29.114,429.919,170.810,30.123,155.665
C09751=1054.307,-28.864,429.905,170.812,30.125,155.666
C09752=1054.313,-28.615,429.892,170.814,30.127,155.666
C09753=1054.319,-28.366,429.879,170.816,30.129,155.666
C09754=1054.324,-28.116,429.865,170.818,30.130,155.666
C09755=1054.331,-27.866,429.851,170.819,30.133,155.666
C09756=1054.337,-27.617,429.838,170.821,30.134,155.667
C09757=1054.343,-27.367,429.825,170.822,30.136,155.667
C09758=1054.350,-27.117,429.812,170.824,30.138,155.667
C09759=1054.356,-26.868,429.798,170.826,30.139,155.667
C09760=1054.362,-26.618,429.784,170.828,30.141,155.668
C09761=1054.368,-26.369,429.771,170.829,30.143,155.668
C09762=1054.375,-26.119,429.758,170.831,30.145,155.668
C09763=1054.380,-25.869,429.744,170.833,30.147,155.668
C09764=1054.387,-25.620,429.730,170.835,30.149,155.668
C09765=1054.393,-25.370,429.717,170.837,30.151,155.669
C09766=1054.399,-25.121,429.703,170.838,30.153,155.669
C09767=1054.405,-24.871,429.690,170.840,30.155,155.669
C09768=1054.411,-24.622,429.676,170.842,30.157,155.669
C09769=1054.417,-24.372,429.662,170.844,30.159,155.670
C09770=1054.424,-24.123,429.649,170.845,30.161,155.670
C09771=1054.429,-23.873,429.635,170.847,30.162,155.670
C09772=1054.436,-23.624,429.621,170.848,30.164,155.670
C09773=1054.442,-23.374,429.607,170.850,30.166,155.670
C09774=1054.448,-23.125,429.594,170.852,30.168,155.671
C09775=1054.455,-22.875,429.580,170.854,30.170,155.671
C09776=1054.461,-22.626,429.567,170.856,30.172,155.671
C09777=1054.466,-22.376,429.553,170.857,30.174,155.671
C09778=1054.473,-22.126,429.539,170.859,30.175,155.672
C09779=1054.479,-21.876,429.525,170.861,30.178,155.672
C09780=1054.485,-21.627,429.512,170.863,30.180,155.672
C09781=1054.492,-21.377,429.498,170.864,30.181,155.672
C09782=1054.497,-21.128,429.484,170.865,30.183,155.673
C09783=1054.504,-20.879,429.471,170.867,30.186,155.673
C09784=1054.511,-20.629,429.457,170.869,30.187,155.673
C09785=1054.516,-20.379,429.443,170.871,30.189,155.673
C09786=1054.522,-20.130,429.430,170.873,30.191,155.673
C09787=1054.528,-19.880,429.416,170.874,30.193,155.674
C09788=1054.535,-19.631,429.402,170.876,30.195,155.674
C09789=1054.541,-19.381,429.387,170.878,30.197,155.674
C09790=1054.547,-19.132,429.374,170.880,30.199,155.674
C09791=1054.554,-18.851,429.358,170.882,30.201,155.675
C09792=1054.561,-18.571,429.344,170.883,30.203,155.675
C09793=1054.568,-18.290,429.327,170.885,30.205,155.675
C09794=1054.575,-18.009,429.311,170.887,30.208,155.676
C09795=1054.581,-17.760,429.298,170.889,30.209,155.676
C09796=1054.588,-17.510,429.285,170.891,30.211,155.676
C09797=1054.594,-17.261,429.270,170.892,30.213,155.676
C09798=1054.600,-17.012,429.257,170.894,30.215,155.676
C09799=1054.606,-16.761,429.242,170.896,30.217,155.677
C09800=1054.613,-16.513,429.228,170.898,30.219,155.677
C09801=1054.619,-16.262,429.214,170.899,30.221,155.677
C09802=1054.625,-16.013,429.201,170.900,30.223,155.677
C09803=1054.632,-15.763,429.187,170.902,30.224,155.678
C09804=1054.638,-15.514,429.173,170.904,30.227,155.678
C09805=1054.644,-15.265,429.159,170.906,30.229,155.678
C09806=1054.650,-15.015,429.145,170.908,30.230,155.678
C09807=1054.656,-14.766,429.131,170.910,30.232,155.679
C09808=1054.663,-14.516,429.117,170.911,30.235,155.679
C09809=1054.668,-14.267,429.102,170.912,30.237,155.679
C09810=1054.675,-14.017,429.089,170.914,30.239,155.679
C09811=1054.681,-13.767,429.075,170.916,30.240,155.680
C09812=1054.687,-13.517,429.060,170.918,30.243,155.680
C09813=1054.693,-13.268,429.047,170.919,30.245,155.680
C09814=1054.699,-13.019,429.032,170.921,30.247,155.680
C09815=1054.705,-12.769,429.018,170.923,30.249,155.681
C09816=1054.711,-12.520,429.005,170.925,30.251,155.681
C09817=1054.718,-12.270,428.990,170.926,30.253,155.681
C09818=1054.723,-12.021,428.976,170.927,30.255,155.681
C09819=1054.730,-11.771,428.961,170.929,30.257,155.682
C09820=1054.736,-11.522,428.948,170.931,30.259,155.682
C09821=1054.742,-11.272,428.933,170.933,30.261,155.682
C09822=1054.748,-11.023,428.919,170.935,30.263,155.682
C09823=1054.755,-10.773,428.904,170.936,30.265,155.683
C09824=1054.760,-10.523,428.890,170.938,30.267,155.683
C09825=1054.767,-10.274,428.876,170.939,30.269,155.683
C09826=1054.773,-10.025,428.862,170.941,30.271,155.683
C09827=1054.779,-9.775,428.847,170.943,30.273,155.684
C09828=1054.785,-9.525,428.833,170.944,30.275,155.684
C09829=1054.792,-9.276,428.819,170.946,30.277,155.684
C09830=1054.797,-9.026,428.805,170.948,30.279,155.685
C09831=1054.804,-8.777,428.790,170.950,30.281,155.685
C09832=1054.811,-8.527,428.776,170.951,30.283,155.685
C09833=1054.816,-8.278,428.762,170.952,30.285,155.685
C09834=1054.823,-8.028,428.747,170.954,30.287,155.686
C09835=1054.829,-7.779,428.734,170.956,30.289,155.686
C09836=1054.835,-7.529,428.719,170.958,30.291,155.686
C09837=1054.841,-7.280,428.705,170.960,30.293,155.686
C09838=1054.847,-7.030,428.690,170.962,30.295,155.687
C09839=1054.854,-6.781,428.676,170.962,30.297,155.687
C09840=1054.860,-6.531,428.662,170.964,30.299,155.687
C09841=1054.866,-6.281,428.647,170.966,30.301,155.687
C09842=1054.873,-6.033,428.633,170.968,30.303,155.688
C09843=1054.879,-5.782,428.619,170.970,30.305,155.688
C09844=1054.885,-5.534,428.604,170.971,30.307,155.688
C09845=1054.891,-5.283,428.590,170.973,30.309,155.688
C09846=1054.898,-5.034,428.576,170.974,30.311,155.689
C09847=1054.904,-4.785,428.561,170.976,30.314,155.689
C09848=1054.910,-4.535,428.546,170.978,30.315,155.689
C09849=1054.916,-4.285,428.532,170.979,30.317,155.689
C09850=1054.923,-4.036,428.518,170.981,30.319,155.690
C09851=1054.929,-3.787,428.503,170.983,30.322,155.690
C09852=1054.934,-3.537,428.489,170.984,30.324,155.690
C09853=1054.941,-3.287,428.474,170.986,30.326,155.691
C09854=1054.947,-3.038,428.459,170.987,30.328,155.691
C09855=1054.955,-2.756,428.443,170.989,30.330,155.691
C09856=1054.961,-2.474,428.426,170.991,30.332,155.691
C09857=1054.968,-2.191,428.410,170.993,30.335,155.692
C09858=1054.975,-1.909,428.394,170.995,30.337,155.692
C09859=1054.980,-1.660,428.379,170.996,30.339,155.692
C09860=1054.987,-1.410,428.364,170.998,30.341,155.693
C09861=1054.993,-1.161,428.349,171.000,30.344,155.693
C09862=1054.999,-0.912,428.335,171.002,30.346,155.693
C09863=1055.005,-0.661,428.320,171.004,30.348,155.694
C09864=1055.011,-0.413,428.306,171.004,30.350,155.694
C09865=1055.017,-0.163,428.291,171.006,30.352,155.694
C09866=1055.024,0.087,428.276,171.008,30.354,155.694
C09867=1055.029,0.336,428.261,171.010,30.356,155.695
C09868=1055.036,0.585,428.246,171.012,30.358,155.695
C09869=1055.042,0.835,428.231,171.012,30.360,155.695
C09870=1055.047,1.085,428.217,171.014,30.363,155.696
C09871=1055.053,1.335,428.202,171.016,30.365,155.696
C09872=1055.060,1.584,428.187,171.018,30.367,155.696
C09873=1055.065,1.833,428.172,171.020,30.370,155.696
C09874=1055.072,2.083,428.158,171.021,30.372,155.697
C09875=1055.078,2.333,428.143,171.022,30.374,155.697
C09876=1055.084,2.582,428.128,171.024,30.376,155.697
C09877=1055.090,2.831,428.113,171.026,30.378,155.698
C09878=1055.097,3.081,428.098,171.028,30.380,155.698
C09879=1055.103,3.330,428.084,171.029,30.382,155.698
C09880=1055.109,3.579,428.069,171.030,30.384,155.698
C09881=1055.115,3.829,428.054,171.032,30.386,155.699
C09882=1055.121,4.078,428.039,171.034,30.389,155.699
C09883=1055.128,4.328,428.024,171.036,30.391,155.699
C09884=1055.134,4.577,428.009,171.037,30.393,155.700
C09885=1055.140,4.827,427.994,171.038,30.395,155.700
C09886=1055.145,5.076,427.979,171.040,30.397,155.700
C09887=1055.152,5.326,427.964,171.042,30.399,155.700
C09888=1055.158,5.576,427.949,171.044,30.401,155.701
C09889=1055.164,5.825,427.935,171.046,30.403,155.701
C09890=1055.170,6.074,427.920,171.046,30.405,155.701
C09891=1055.177,6.324,427.905,171.048,30.408,155.702
C09892=1055.183,6.574,427.890,171.050,30.410,155.702
C09893=1055.189,6.822,427.875,171.052,30.412,155.702
C09894=1055.195,7.072,427.860,171.054,30.414,155.702
C09895=1055.202,7.322,427.845,171.055,30.416,155.703
C09896=1055.208,7.571,427.830,171.056,30.418,155.703
C09897=1055.214,7.821,427.815,171.058,30.420,155.703
C09898=1055.219,8.070,427.800,171.060,30.422,155.704
C09899=1055.226,8.319,427.785,171.062,30.425,155.704
C09900=1055.232,8.569,427.770,171.063,30.427,155.704
C09901=1055.239,8.819,427.755,171.064,30.429,155.705
C09902=1055.245,9.068,427.740,171.066,30.431,155.705
C09903=1055.251,9.317,427.725,171.068,30.434,155.705
C09904=1055.257,9.567,427.710,171.070,30.436,155.705
C09905=1055.264,9.817,427.695,171.071,30.438,155.706
C09906=1055.269,10.067,427.680,171.072,30.440,155.706
C09907=1055.276,10.316,427.664,171.074,30.442,155.706
C09908=1055.282,10.565,427.649,171.076,30.444,155.707
C09909=1055.288,10.814,427.634,171.078,30.446,155.707
C09910=1055.295,11.064,427.620,171.079,30.448,155.707
C09911=1055.301,11.314,427.605,171.080,30.450,155.707
C09912=1055.308,11.563,427.589,171.082,30.453,155.708
C09913=1055.313,11.813,427.573,171.084,30.455,155.708
C09914=1055.320,12.062,427.558,171.086,30.457,155.708
C09915=1055.326,12.311,427.544,171.088,30.459,155.709
C09916=1055.332,12.560,427.528,171.088,30.461,155.709
C09917=1055.339,12.810,427.513,171.090,30.463,155.709
C09918=1055.345,13.060,427.498,171.092,30.465,155.709
C09919=1055.352,13.344,427.481,171.094,30.468,155.710
C09920=1055.359,13.628,427.463,171.096,30.470,155.710
C09921=1055.367,13.912,427.446,171.097,30.473,155.711
C09922=1055.373,14.196,427.429,171.099,30.475,155.711
C09923=1055.380,14.445,427.414,171.101,30.477,155.711
C09924=1055.386,14.695,427.398,171.103,30.479,155.711
C09925=1055.392,14.945,427.383,171.104,30.482,155.712
C09926=1055.398,15.194,427.367,171.105,30.484,155.712
C09927=1055.404,15.444,427.352,171.107,30.486,155.712
C09928=1055.411,15.693,427.337,171.109,30.488,155.713
C09929=1055.417,15.943,427.321,171.110,30.490,155.713
C09930=1055.422,16.192,427.306,171.112,30.492,155.713
C09931=1055.429,16.441,427.291,171.113,30.495,155.714
C09932=1055.435,16.691,427.275,171.115,30.497,155.714
C09933=1055.441,16.940,427.260,171.117,30.499,155.714
C09934=1055.447,17.190,427.244,171.118,30.501,155.714
C09935=1055.453,17.439,427.229,171.120,30.504,155.715
C09936=1055.460,17.689,427.214,171.121,30.506,155.715
C09937=1055.466,17.938,427.198,171.123,30.508,155.715
C09938=1055.472,18.188,427.183,171.124,30.510,155.716
C09939=1055.478,18.437,427.166,171.126,30.513,155.716
C09940=1055.484,18.686,427.152,171.128,30.515,155.716
C09941=1055.491,18.935,427.136,171.130,30.517,155.717
C09942=1055.496,19.185,427.121,171.131,30.520,155.717
C09943=1055.503,19.434,427.105,171.132,30.522,155.717
C09944=1055.509,19.684,427.089,171.134,30.524,155.718
C09945=1055.515,19.933,427.074,171.136,30.526,155.718
C09946=1055.522,20.183,427.059,171.138,30.528,155.718
C09947=1055.528,20.432,427.043,171.138,30.530,155.719
C09948=1055.534,20.682,427.028,171.140,30.533,155.719
C09949=1055.540,20.931,427.011,171.142,30.535,155.719
C09950=1055.546,21.181,426.996,171.144,30.537,155.719
C09951=1055.552,21.430,426.980,171.145,30.539,155.720
C09952=1055.558,21.680,426.965,171.146,30.542,155.720
C09953=1055.565,21.929,426.949,171.148,30.544,155.720
C09954=1055.570,22.179,426.933,171.150,30.546,155.721
C09955=1055.576,22.428,426.918,171.151,30.548,155.721
C09956=1055.582,22.677,426.902,171.153,30.551,155.721
C09957=1055.589,22.927,426.887,171.154,30.553,155.722
C09958=1055.595,23.176,426.871,171.156,30.555,155.722
C09959=1055.601,23.426,426.856,171.157,30.557,155.722
C09960=1055.607,23.675,426.839,171.159,30.560,155.723
C09961=1055.614,23.924,426.824,171.161,30.562,155.723
C09962=1055.619,24.174,426.808,171.163,30.564,155.723
C09963=1055.625,24.423,426.792,171.163,30.566,155.724
C09964=1055.632,24.672,426.776,171.165,30.569,155.724
C09965=1055.638,24.922,426.761,171.167,30.571,155.724
C09966=1055.644,25.171,426.745,171.169,30.573,155.725
C09967=1055.650,25.421,426.729,171.170,30.575,155.725
C09968=1055.657,25.670,426.714,171.171,30.577,155.725
C09969=1055.663,25.920,426.698,171.173,30.580,155.726
C09970=1055.669,26.169,426.682,171.175,30.582,155.726
C09971=1055.675,26.419,426.666,171.177,30.584,155.726
C09972=1055.681,26.668,426.650,171.178,30.586,155.726
C09973=1055.687,26.917,426.635,171.179,30.589,155.727
C09974=1055.694,27.168,426.619,171.181,30.591,155.727
C09975=1055.700,27.417,426.603,171.183,30.593,155.727
C09976=1055.706,27.666,426.587,171.184,30.595,155.728
C09977=1055.712,27.915,426.570,171.186,30.598,155.728
C09978=1055.719,28.165,426.556,171.188,30.600,155.728
C09979=1055.725,28.414,426.539,171.189,30.602,155.729
C09980=1055.731,28.664,426.523,171.190,30.604,155.729
C09981=1055.737,28.913,426.507,171.192,30.606,155.729
C09982=1055.743,29.162,426.491,171.194,30.609,155.730
C09983=1055.750,29.448,426.473,171.196,30.611,155.730
C09984=1055.757,29.733,426.455,171.197,30.614,155.730
C09985=1055.764,30.019,426.436,171.199,30.617,155.731
C09986=1055.770,30.304,426.418,171.201,30.620,155.731
C09987=1055.777,30.553,426.402,171.202,30.622,155.732
C09988=1055.783,30.803,426.386,171.204,30.624,155.732
C09989=1055.789,31.052,426.370,171.205,30.626,155.732
C09990=1055.795,31.301,426.354,171.207,30.628,155.732
C09991=1055.801,31.551,426.337,171.208,30.631,155.733
C09992=1055.807,31.800,426.322,171.210,30.633,155.733
C09993=1055.814,32.050,426.306,171.212,30.635,155.733
C09994=1055.820,32.300,426.289,171.213,30.638,155.734
C09995=1055.826,32.549,426.273,171.214,30.640,155.734
C09996=1055.832,32.798,426.257,171.216,30.642,155.734
//INST
///DATE 2021/06/25 14:46
///ATTR SC,RW,RJ
////FRAME ROBOT
///GROUP1 RB1
NOP
MOVL C00000 V=800.0 PL=0
MOVL C00001 V=800.0 PL=0
MOVL C00002 V=800.0 PL=0
MOVL C00003 V=800.0 PL=0
MOVL C00004 V=800.0 PL=0
MOVL C00005 V=800.0 PL=0
MOVL C00006 V=800.0 PL=0
MOVL C00007 V=800.0 PL=0
MOVL C00008 V=800.0 PL=0
MOVL C00009 V=800.0 PL=0
MOVL C00010 V=800.0 PL=0
MOVL C00011 V=800.0 PL=0
MOVL C00012 V=800.0 PL=0
MOVL C00013 V=800.0 PL=0
MOVL C00014 V=800.0 PL=0
MOVL C00015 V=800.0 PL=0
MOVL C00016 V=800.0 PL=0
MOVL C00017 V=800.0 PL=0
MOVL C00018 V=800.0 PL=0
MOVL C00019 V=800.0 PL=0
MOVL C00020 V=800.0 PL=0
MOVL C00021 V=800.0 PL=0
MOVL C00022 V=800.0 PL=0
MOVL C00023 V=800.0 PL=0
MOVL C00024 V=800.0 PL=0
MOVL C00025 V=800.0 PL=0
MOVL C00026 V=800.0 PL=0
MOVL C00027 V=800.0 PL=0
MOVL C00028 V=800.0 PL=0
MOVL C00029 V=800.0 PL=0
MOVL C00030 V=800.0 PL=0
MOVL C00031 V=800.0 PL=0
MOVL C00032 V=800.0 PL=0
MOVL C00033 V=800.0 PL=0
MOVL C00034 V=800.0 PL=0
MOVL C00035 V=800.0 PL=0
MOVL C00036 V=800.0 PL=0
MOVL C00037 V=800.0 PL=0
MOVL C00038 V=800.0 PL=0
MOVL C00039 V=800.0 PL=0
MOVL C00040 V=800.0 PL=0
MOVL C00041 V=800.0 PL=0
MOVL C00042 V=800.0 PL=0
MOVL C00043 V=800.0 PL=0
MOVL C00044 V=800.0 PL=0
MOVL C00045 V=800.0 PL=0
MOVL C00046 V=800.0 PL=0
MOVL C00047 V=800.0 PL=0
MOVL C00048 V=800.0 PL=0
MOVL C00049 V=800.0 PL=0
MOVL C00050 V=800.0 PL=0
MOVL C00051 V=800.0 PL=0
MOVL C00052 V=800.0 PL=0
MOVL C00053 V=800.0 PL=0
MOVL C00054 V=800.0 PL=0
MOVL C00055 V=800.0 PL=0
MOVL C00056 V=800.0 PL=0
MOVL C00057 V=800.0 PL=0
MOVL C00058 V=800.0 PL=0
MOVL C00059 V=800.0 PL=0
MOVL C00060 V=800.0 PL=0
MOVL C00061 V=800.0 PL=0
MOVL C00062 V=800.0 PL=0
MOVL C00063 V=800.0 PL=0
MOVL C00064 V=800.0 PL=0
MOVL C00065 V=800.0 PL=0
MOVL C00066 V=800.0 PL=0
MOVL C00067 V=800.0 PL=0
MOVL C00068 V=800.0 PL=0
MOVL C00069 V=800.0 PL=0
MOVL C00070 V=800.0 PL=0
MOVL C00071 V=800.0 PL=0
MOVL C00072 V=800.0 PL=0
MOVL C00073 V=800.0 PL=0
MOVL C00074 V=800.0 PL=0
MOVL C00075 V=800.0 PL=0
MOVL C00076 V=800.0 PL=0
MOVL C00077 V=800.0 PL=0
MOVL C00078 V=800.0 PL=0
MOVL C00079 V=800.0 PL=0
MOVL C00080 V=800.0 PL=0
MOVL C00081 V=800.0 PL=0
MOVL C00082 V=800.0 PL=0
MOVL C00083 V=800.0 PL=0
MOVL C00084 V=800.0 PL=0
MOVL C00085 V=800.0 PL=0
MOVL C00086 V=800.0 PL=0
MOVL C00087 V=800.0 PL=0
MOVL C00088 V=800.0 PL=0
MOVL C00089 V=800.0 PL=0
MOVL C00090 V=800.0 PL=0
MOVL C00091 V=800.0 PL=0
MOVL C00092 V=800.0 PL=0
MOVL C00093 V=800.0 PL=0
MOVL C00094 V=800.0 PL=0
MOVL C00095 V=800.0 PL=0
MOVL C00096 V=800.0 PL=0
MOVL C00097 V=800.0 PL=0
MOVL C00098 V=800.0 PL=0
MOVL C00099 V=800.0 PL=0
MOVL C00100 V=800.0 PL=0
MOVL C00101 V=800.0 PL=0
MOVL C00102 V=800.0 PL=0
MOVL C00103 V=800.0 PL=0
MOVL C00104 V=800.0 PL=0
MOVL C00105 V=800.0 PL=0
MOVL C00106 V=800.0 PL=0
MOVL C00107 V=800.0 PL=0
MOVL C00108 V=800.0 PL=0
MOVL C00109 V=800.0 PL=0
MOVL C00110 V=800.0 PL=0
MOVL C00111 V=800.0 PL=0
MOVL C00112 V=800.0 PL=0
MOVL C00113 V=800.0 PL=0
MOVL C00114 V=800.0 PL=0
MOVL C00115 V=800.0 PL=0
MOVL C00116 V=800.0 PL=0
MOVL C00117 V=800.0 PL=0
MOVL C00118 V=800.0 PL=0
MOVL C00119 V=800.0 PL=0
MOVL C00120 V=800.0 PL=0
MOVL C00121 V=800.0 PL=0
MOVL C00122 V=800.0 PL=0
MOVL C00123 V=800.0 PL=0
MOVL C00124 V=800.0 PL=0
MOVL C00125 V=800.0 PL=0
MOVL C00126 V=800.0 PL=0
MOVL C00127 V=800.0 PL=0
MOVL C00128 V=800.0 PL=0
MOVL C00129 V=800.0 PL=0
MOVL C00130 V=800.0 PL=0
MOVL C00131 V=800.0 PL=0
MOVL C00132 V=800.0 PL=0
MOVL C00133 V=800.0 PL=0
MOVL C00134 V=800.0 PL=0
MOVL C00135 V=800.0 PL=0
MOVL C00136 V=800.0 PL=0
MOVL C00137 V=800.0 PL=0
MOVL C00138 V=800.0 PL=0
MOVL C00139 V=800.0 PL=0
MOVL C00140 V=800.0 PL=0
MOVL C00141 V=800.0 PL=0
MOVL C00142 V=800.0 PL=0
MOVL C00143 V=800.0 PL=0
MOVL C00144 V=800.0 PL=0
MOVL C00145 V=800.0 PL=0
MOVL C00146 V=800.0 PL=0
MOVL C00147 V=800.0 PL=0
MOVL C00148 V=800.0 PL=0
MOVL C00149 V=800.0 PL=0
MOVL C00150 V=800.0 PL=0
MOVL C00151 V=800.0 PL=0
MOVL C00152 V=800.0 PL=0
MOVL C00153 V=800.0 PL=0
MOVL C00154 V=800.0 PL=0
MOVL C00155 V=800.0 PL=0
MOVL C00156 V=800.0 PL=0
MOVL C00157 V=800.0 PL=0
MOVL C00158 V=800.0 PL=0
MOVL C00159 V=800.0 PL=0
MOVL C00160 V=800.0 PL=0
MOVL C00161 V=800.0 PL=0
MOVL C00162 V=800.0 PL=0
MOVL C00163 V=800.0 PL=0
MOVL C00164 V=800.0 PL=0
MOVL C00165 V=800.0 PL=0
MOVL C00166 V=800.0 PL=0
MOVL C00167 V=800.0 PL=0
MOVL C00168 V=800.0 PL=0
MOVL C00169 V=800.0 PL=0
MOVL C00170 V=800.0 PL=0
MOVL C00171 V=800.0 PL=0
MOVL C00172 V=800.0 PL=0
MOVL C00173 V=800.0 PL=0
MOVL C00174 V=800.0 PL=0
MOVL C00175 V=800.0 PL=0
MOVL C00176 V=800.0 PL=0
MOVL C00177 V=800.0 PL=0
MOVL C00178 V=800.0 PL=0
MOVL C00179 V=800.0 PL=0
MOVL C00180 V=800.0 PL=0
MOVL C00181 V=800.0 PL=0
MOVL C00182 V=800.0 PL=0
MOVL C00183 V=800.0 PL=0
MOVL C00184 V=800.0 PL=0
MOVL C00185 V=800.0 PL=0
MOVL C00186 V=800.0 PL=0
MOVL C00187 V=800.0 PL=0
MOVL C00188 V=800.0 PL=0
MOVL C00189 V=800.0 PL=0
MOVL C00190 V=800.0 PL=0
MOVL C00191 V=800.0 PL=0
MOVL C00192 V=800.0 PL=0
MOVL C00193 V=800.0 PL=0
MOVL C00194 V=800.0 PL=0
MOVL C00195 V=800.0 PL=0
MOVL C00196 V=800.0 PL=0
MOVL C00197 V=800.0 PL=0
MOVL C00198 V=800.0 PL=0
MOVL C00199 V=800.0 PL=0
MOVL C00200 V=800.0 PL=0
MOVL C00201 V=800.0 PL=0
MOVL C00202 V=800.0 PL=0
MOVL C00203 V=800.0 PL=0
MOVL C00204 V=800.0 PL=0
MOVL C00205 V=800.0 PL=0
MOVL C00206 V=800.0 PL=0
MOVL C00207 V=800.0 PL=0
MOVL C00208 V=800.0 PL=0
MOVL C00209 V=800.0 PL=0
MOVL C00210 V=800.0 PL=0
MOVL C00211 V=800.0 PL=0
MOVL C00212 V=800.0 PL=0
MOVL C00213 V=800.0 PL=0
MOVL C00214 V=800.0 PL=0
MOVL C00215 V=800.0 PL=0
MOVL C00216 V=800.0 PL=0
MOVL C00217 V=800.0 PL=0
MOVL C00218 V=800.0 PL=0
MOVL C00219 V=800.0 PL=0
MOVL C00220 V=800.0 PL=0
MOVL C00221 V=800.0 PL=0
MOVL C00222 V=800.0 PL=0
MOVL C00223 V=800.0 PL=0
MOVL C00224 V=800.0 PL=0
MOVL C00225 V=800.0 PL=0
MOVL C00226 V=800.0 PL=0
MOVL C00227 V=800.0 PL=0
MOVL C00228 V=800.0 PL=0
MOVL C00229 V=800.0 PL=0
MOVL C00230 V=800.0 PL=0
MOVL C00231 V=800.0 PL=0
MOVL C00232 V=800.0 PL=0
MOVL C00233 V=800.0 PL=0
MOVL C00234 V=800.0 PL=0
MOVL C00235 V=800.0 PL=0
MOVL C00236 V=800.0 PL=0
MOVL C00237 V=800.0 PL=0
MOVL C00238 V=800.0 PL=0
MOVL C00239 V=800.0 PL=0
MOVL C00240 V=800.0 PL=0
MOVL C00241 V=800.0 PL=0
MOVL C00242 V=800.0 PL=0
MOVL C00243 V=800.0 PL=0
MOVL C00244 V=800.0 PL=0
MOVL C00245 V=800.0 PL=0
MOVL C00246 V=800.0 PL=0
MOVL C00247 V=800.0 PL=0
MOVL C00248 V=800.0 PL=0
MOVL C00249 V=800.0 PL=0
MOVL C00250 V=800.0 PL=0
MOVL C00251 V=800.0 PL=0
MOVL C00252 V=800.0 PL=0
MOVL C00253 V=800.0 PL=0
MOVL C00254 V=800.0 PL=0
MOVL C00255 V=800.0 PL=0
MOVL C00256 V=800.0 PL=0
MOVL C00257 V=800.0 PL=0
MOVL C00258 V=800.0 PL=0
MOVL C00259 V=800.0 PL=0
MOVL C00260 V=800.0 PL=0
MOVL C00261 V=800.0 PL=0
MOVL C00262 V=800.0 PL=0
MOVL C00263 V=800.0 PL=0
MOVL C00264 V=800.0 PL=0
MOVL C00265 V=800.0 PL=0
MOVL C00266 V=800.0 PL=0
MOVL C00267 V=800.0 PL=0
MOVL C00268 V=800.0 PL=0
MOVL C00269 V=800.0 PL=0
MOVL C00270 V=800.0 PL=0
MOVL C00271 V=800.0 PL=0
MOVL C00272 V=800.0 PL=0
MOVL C00273 V=800.0 PL=0
MOVL C00274 V=800.0 PL=0
MOVL C00275 V=800.0 PL=0
MOVL C00276 V=800.0 PL=0
MOVL C00277 V=800.0 PL=0
MOVL C00278 V=800.0 PL=0
MOVL C00279 V=800.0 PL=0
MOVL C00280 V=800.0 PL=0
MOVL C00281 V=800.0 PL=0
MOVL C00282 V=800.0 PL=0
MOVL C00283 V=800.0 PL=0
MOVL C00284 V=800.0 PL=0
MOVL C00285 V=800.0 PL=0
MOVL C00286 V=800.0 PL=0
MOVL C00287 V=800.0 PL=0
MOVL C00288 V=800.0 PL=0
MOVL C00289 V=800.0 PL=0
MOVL C00290 V=800.0 PL=0
MOVL C00291 V=800.0 PL=0
MOVL C00292 V=800.0 PL=0
MOVL C00293 V=800.0 PL=0
MOVL C00294 V=800.0 PL=0
MOVL C00295 V=800.0 PL=0
MOVL C00296 V=800.0 PL=0
MOVL C00297 V=800.0 PL=0
MOVL C00298 V=800.0 PL=0
MOVL C00299 V=800.0 PL=0
MOVL C00300 V=800.0 PL=0
MOVL C00301 V=800.0 PL=0
MOVL C00302 V=800.0 PL=0
MOVL C00303 V=800.0 PL=0
MOVL C00304 V=800.0 PL=0
MOVL C00305 V=800.0 PL=0
MOVL C00306 V=800.0 PL=0
MOVL C00307 V=800.0 PL=0
MOVL C00308 V=800.0 PL=0
MOVL C00309 V=800.0 PL=0
MOVL C00310 V=800.0 PL=0
MOVL C00311 V=800.0 PL=0
MOVL C00312 V=800.0 PL=0
MOVL C00313 V=800.0 PL=0
MOVL C00314 V=800.0 PL=0
MOVL C00315 V=800.0 PL=0
MOVL C00316 V=800.0 PL=0
MOVL C00317 V=800.0 PL=0
MOVL C00318 V=800.0 PL=0
MOVL C00319 V=800.0 PL=0
MOVL C00320 V=800.0 PL=0
MOVL C00321 V=800.0 PL=0
MOVL C00322 V=800.0 PL=0
MOVL C00323 V=800.0 PL=0
MOVL C00324 V=800.0 PL=0
MOVL C00325 V=800.0 PL=0
MOVL C00326 V=800.0 PL=0
MOVL C00327 V=800.0 PL=0
MOVL C00328 V=800.0 PL=0
MOVL C00329 V=800.0 PL=0
MOVL C00330 V=800.0 PL=0
MOVL C00331 V=800.0 PL=0
MOVL C00332 V=800.0 PL=0
MOVL C00333 V=800.0 PL=0
MOVL C00334 V=800.0 PL=0
MOVL C00335 V=800.0 PL=0
MOVL C00336 V=800.0 PL=0
MOVL C00337 V=800.0 PL=0
MOVL C00338 V=800.0 PL=0
MOVL C00339 V=800.0 PL=0
MOVL C00340 V=800.0 PL=0
MOVL C00341 V=800.0 PL=0
MOVL C00342 V=800.0 PL=0
MOVL C00343 V=800.0 PL=0
MOVL C00344 V=800.0 PL=0
MOVL C00345 V=800.0 PL=0
MOVL C00346 V=800.0 PL=0
MOVL C00347 V=800.0 PL=0
MOVL C00348 V=800.0 PL=0
MOVL C00349 V=800.0 PL=0
MOVL C00350 V=800.0 PL=0
MOVL C00351 V=800.0 PL=0
MOVL C00352 V=800.0 PL=0
MOVL C00353 V=800.0 PL=0
MOVL C00354 V=800.0 PL=0
MOVL C00355 V=800.0 PL=0
MOVL C00356 V=800.0 PL=0
MOVL C00357 V=800.0 PL=0
MOVL C00358 V=800.0 PL=0
MOVL C00359 V=800.0 PL=0
MOVL C00360 V=800.0 PL=0
MOVL C00361 V=800.0 PL=0
MOVL C00362 V=800.0 PL=0
MOVL C00363 V=800.0 PL=0
MOVL C00364 V=800.0 PL=0
MOVL C00365 V=800.0 PL=0
MOVL C00366 V=800.0 PL=0
MOVL C00367 V=800.0 PL=0
MOVL C00368 V=800.0 PL=0
MOVL C00369 V=800.0 PL=0
MOVL C00370 V=800.0 PL=0
MOVL C00371 V=800.0 PL=0
MOVL C00372 V=800.0 PL=0
MOVL C00373 V=800.0 PL=0
MOVL C00374 V=800.0 PL=0
MOVL C00375 V=800.0 PL=0
MOVL C00376 V=800.0 PL=0
MOVL C00377 V=800.0 PL=0
MOVL C00378 V=800.0 PL=0
MOVL C00379 V=800.0 PL=0
MOVL C00380 V=800.0 PL=0
MOVL C00381 V=800.0 PL=0
MOVL C00382 V=800.0 PL=0
MOVL C00383 V=800.0 PL=0
MOVL C00384 V=800.0 PL=0
MOVL C00385 V=800.0 PL=0
MOVL C00386 V=800.0 PL=0
MOVL C00387 V=800.0 PL=0
MOVL C00388 V=800.0 PL=0
MOVL C00389 V=800.0 PL=0
MOVL C00390 V=800.0 PL=0
MOVL C00391 V=800.0 PL=0
MOVL C00392 V=800.0 PL=0
MOVL C00393 V=800.0 PL=0
MOVL C00394 V=800.0 PL=0
MOVL C00395 V=800.0 PL=0
MOVL C00396 V=800.0 PL=0
MOVL C00397 V=800.0 PL=0
MOVL C00398 V=800.0 PL=0
MOVL C00399 V=800.0 PL=0
MOVL C00400 V=800.0 PL=0
MOVL C00401 V=800.0 PL=0
MOVL C00402 V=800.0 PL=0
MOVL C00403 V=800.0 PL=0
MOVL C00404 V=800.0 PL=0
MOVL C00405 V=800.0 PL=0
MOVL C00406 V=800.0 PL=0
MOVL C00407 V=800.0 PL=0
MOVL C00408 V=800.0 PL=0
MOVL C00409 V=800.0 PL=0
MOVL C00410 V=800.0 PL=0
MOVL C00411 V=800.0 PL=0
MOVL C00412 V=800.0 PL=0
MOVL C00413 V=800.0 PL=0
MOVL C00414 V=800.0 PL=0
MOVL C00415 V=800.0 PL=0
MOVL C00416 V=800.0 PL=0
MOVL C00417 V=800.0 PL=0
MOVL C00418 V=800.0 PL=0
MOVL C00419 V=800.0 PL=0
MOVL C00420 V=800.0 PL=0
MOVL C00421 V=800.0 PL=0
MOVL C00422 V=800.0 PL=0
MOVL C00423 V=800.0 PL=0
MOVL C00424 V=800.0 PL=0
MOVL C00425 V=800.0 PL=0
MOVL C00426 V=800.0 PL=0
MOVL C00427 V=800.0 PL=0
MOVL C00428 V=800.0 PL=0
MOVL C00429 V=800.0 PL=0
MOVL C00430 V=800.0 PL=0
MOVL C00431 V=800.0 PL=0
MOVL C00432 V=800.0 PL=0
MOVL C00433 V=800.0 PL=0
MOVL C00434 V=800.0 PL=0
MOVL C00435 V=800.0 PL=0
MOVL C00436 V=800.0 PL=0
MOVL C00437 V=800.0 PL=0
MOVL C00438 V=800.0 PL=0
MOVL C00439 V=800.0 PL=0
MOVL C00440 V=800.0 PL=0
MOVL C00441 V=800.0 PL=0
MOVL C00442 V=800.0 PL=0
MOVL C00443 V=800.0 PL=0
MOVL C00444 V=800.0 PL=0
MOVL C00445 V=800.0 PL=0
MOVL C00446 V=800.0 PL=0
MOVL C00447 V=800.0 PL=0
MOVL C00448 V=800.0 PL=0
MOVL C00449 V=800.0 PL=0
MOVL C00450 V=800.0 PL=0
MOVL C00451 V=800.0 PL=0
MOVL C00452 V=800.0 PL=0
MOVL C00453 V=800.0 PL=0
MOVL C00454 V=800.0 PL=0
MOVL C00455 V=800.0 PL=0
MOVL C00456 V=800.0 PL=0
MOVL C00457 V=800.0 PL=0
MOVL C00458 V=800.0 PL=0
MOVL C00459 V=800.0 PL=0
MOVL C00460 V=800.0 PL=0
MOVL C00461 V=800.0 PL=0
MOVL C00462 V=800.0 PL=0
MOVL C00463 V=800.0 PL=0
MOVL C00464 V=800.0 PL=0
MOVL C00465 V=800.0 PL=0
MOVL C00466 V=800.0 PL=0
MOVL C00467 V=800.0 PL=0
MOVL C00468 V=800.0 PL=0
MOVL C00469 V=800.0 PL=0
MOVL C00470 V=800.0 PL=0
MOVL C00471 V=800.0 PL=0
MOVL C00472 V=800.0 PL=0
MOVL C00473 V=800.0 PL=0
MOVL C00474 V=800.0 PL=0
MOVL C00475 V=800.0 PL=0
MOVL C00476 V=800.0 PL=0
MOVL C00477 V=800.0 PL=0
MOVL C00478 V=800.0 PL=0
MOVL C00479 V=800.0 PL=0
MOVL C00480 V=800.0 PL=0
MOVL C00481 V=800.0 PL=0
MOVL C00482 V=800.0 PL=0
MOVL C00483 V=800.0 PL=0
MOVL C00484 V=800.0 PL=0
MOVL C00485 V=800.0 PL=0
MOVL C00486 V=800.0 PL=0
MOVL C00487 V=800.0 PL=0
MOVL C00488 V=800.0 PL=0
MOVL C00489 V=800.0 PL=0
MOVL C00490 V=800.0 PL=0
MOVL C00491 V=800.0 PL=0
MOVL C00492 V=800.0 PL=0
MOVL C00493 V=800.0 PL=0
MOVL C00494 V=800.0 PL=0
MOVL C00495 V=800.0 PL=0
MOVL C00496 V=800.0 PL=0
MOVL C00497 V=800.0 PL=0
MOVL C00498 V=800.0 PL=0
MOVL C00499 V=800.0 PL=0
MOVL C00500 V=800.0 PL=0
MOVL C00501 V=800.0 PL=0
MOVL C00502 V=800.0 PL=0
MOVL C00503 V=800.0 PL=0
MOVL C00504 V=800.0 PL=0
MOVL C00505 V=800.0 PL=0
MOVL C00506 V=800.0 PL=0
MOVL C00507 V=800.0 PL=0
MOVL C00508 V=800.0 PL=0
MOVL C00509 V=800.0 PL=0
MOVL C00510 V=800.0 PL=0
MOVL C00511 V=800.0 PL=0
MOVL C00512 V=800.0 PL=0
MOVL C00513 V=800.0 PL=0
MOVL C00514 V=800.0 PL=0
MOVL C00515 V=800.0 PL=0
MOVL C00516 V=800.0 PL=0
MOVL C00517 V=800.0 PL=0
MOVL C00518 V=800.0 PL=0
MOVL C00519 V=800.0 PL=0
MOVL C00520 V=800.0 PL=0
MOVL C00521 V=800.0 PL=0
MOVL C00522 V=800.0 PL=0
MOVL C00523 V=800.0 PL=0
MOVL C00524 V=800.0 PL=0
MOVL C00525 V=800.0 PL=0
MOVL C00526 V=800.0 PL=0
MOVL C00527 V=800.0 PL=0
MOVL C00528 V=800.0 PL=0
MOVL C00529 V=800.0 PL=0
MOVL C00530 V=800.0 PL=0
MOVL C00531 V=800.0 PL=0
MOVL C00532 V=800.0 PL=0
MOVL C00533 V=800.0 PL=0
MOVL C00534 V=800.0 PL=0
MOVL C00535 V=800.0 PL=0
MOVL C00536 V=800.0 PL=0
MOVL C00537 V=800.0 PL=0
MOVL C00538 V=800.0 PL=0
MOVL C00539 V=800.0 PL=0
MOVL C00540 V=800.0 PL=0
MOVL C00541 V=800.0 PL=0
MOVL C00542 V=800.0 PL=0
MOVL C00543 V=800.0 PL=0
MOVL C00544 V=800.0 PL=0
MOVL C00545 V=800.0 PL=0
MOVL C00546 V=800.0 PL=0
MOVL C00547 V=800.0 PL=0
MOVL C00548 V=800.0 PL=0
MOVL C00549 V=800.0 PL=0
MOVL C00550 V=800.0 PL=0
MOVL C00551 V=800.0 PL=0
MOVL C00552 V=800.0 PL=0
MOVL C00553 V=800.0 PL=0
MOVL C00554 V=800.0 PL=0
MOVL C00555 V=800.0 PL=0
MOVL C00556 V=800.0 PL=0
MOVL C00557 V=800.0 PL=0
MOVL C00558 V=800.0 PL=0
MOVL C00559 V=800.0 PL=0
MOVL C00560 V=800.0 PL=0
MOVL C00561 V=800.0 PL=0
MOVL C00562 V=800.0 PL=0
MOVL C00563 V=800.0 PL=0
MOVL C00564 V=800.0 PL=0
MOVL C00565 V=800.0 PL=0
MOVL C00566 V=800.0 PL=0
MOVL C00567 V=800.0 PL=0
MOVL C00568 V=800.0 PL=0
MOVL C00569 V=800.0 PL=0
MOVL C00570 V=800.0 PL=0
MOVL C00571 V=800.0 PL=0
MOVL C00572 V=800.0 PL=0
MOVL C00573 V=800.0 PL=0
MOVL C00574 V=800.0 PL=0
MOVL C00575 V=800.0 PL=0
MOVL C00576 V=800.0 PL=0
MOVL C00577 V=800.0 PL=0
MOVL C00578 V=800.0 PL=0
MOVL C00579 V=800.0 PL=0
MOVL C00580 V=800.0 PL=0
MOVL C00581 V=800.0 PL=0
MOVL C00582 V=800.0 PL=0
MOVL C00583 V=800.0 PL=0
MOVL C00584 V=800.0 PL=0
MOVL C00585 V=800.0 PL=0
MOVL C00586 V=800.0 PL=0
MOVL C00587 V=800.0 PL=0
MOVL C00588 V=800.0 PL=0
MOVL C00589 V=800.0 PL=0
MOVL C00590 V=800.0 PL=0
MOVL C00591 V=800.0 PL=0
MOVL C00592 V=800.0 PL=0
MOVL C00593 V=800.0 PL=0
MOVL C00594 V=800.0 PL=0
MOVL C00595 V=800.0 PL=0
MOVL C00596 V=800.0 PL=0
MOVL C00597 V=800.0 PL=0
MOVL C00598 V=800.0 PL=0
MOVL C00599 V=800.0 PL=0
MOVL C00600 V=800.0 PL=0
MOVL C00601 V=800.0 PL=0
MOVL C00602 V=800.0 PL=0
MOVL C00603 V=800.0 PL=0
MOVL C00604 V=800.0 PL=0
MOVL C00605 V=800.0 PL=0
MOVL C00606 V=800.0 PL=0
MOVL C00607 V=800.0 PL=0
MOVL C00608 V=800.0 PL=0
MOVL C00609 V=800.0 PL=0
MOVL C00610 V=800.0 PL=0
MOVL C00611 V=800.0 PL=0
MOVL C00612 V=800.0 PL=0
MOVL C00613 V=800.0 PL=0
MOVL C00614 V=800.0 PL=0
MOVL C00615 V=800.0 PL=0
MOVL C00616 V=800.0 PL=0
MOVL C00617 V=800.0 PL=0
MOVL C00618 V=800.0 PL=0
MOVL C00619 V=800.0 PL=0
MOVL C00620 V=800.0 PL=0
MOVL C00621 V=800.0 PL=0
MOVL C00622 V=800.0 PL=0
MOVL C00623 V=800.0 PL=0
MOVL C00624 V=800.0 PL=0
MOVL C00625 V=800.0 PL=0
MOVL C00626 V=800.0 PL=0
MOVL C00627 V=800.0 PL=0
MOVL C00628 V=800.0 PL=0
MOVL C00629 V=800.0 PL=0
MOVL C00630 V=800.0 PL=0
MOVL C00631 V=800.0 PL=0
MOVL C00632 V=800.0 PL=0
MOVL C00633 V=800.0 PL=0
MOVL C00634 V=800.0 PL=0
MOVL C00635 V=800.0 PL=0
MOVL C00636 V=800.0 PL=0
MOVL C00637 V=800.0 PL=0
MOVL C00638 V=800.0 PL=0
MOVL C00639 V=800.0 PL=0
MOVL C00640 V=800.0 PL=0
MOVL C00641 V=800.0 PL=0
MOVL C00642 V=800.0 PL=0
MOVL C00643 V=800.0 PL=0
MOVL C00644 V=800.0 PL=0
MOVL C00645 V=800.0 PL=0
MOVL C00646 V=800.0 PL=0
MOVL C00647 V=800.0 PL=0
MOVL C00648 V=800.0 PL=0
MOVL C00649 V=800.0 PL=0
MOVL C00650 V=800.0 PL=0
MOVL C00651 V=800.0 PL=0
MOVL C00652 V=800.0 PL=0
MOVL C00653 V=800.0 PL=0
MOVL C00654 V=800.0 PL=0
MOVL C00655 V=800.0 PL=0
MOVL C00656 V=800.0 PL=0
MOVL C00657 V=800.0 PL=0
MOVL C00658 V=800.0 PL=0
MOVL C00659 V=800.0 PL=0
MOVL C00660 V=800.0 PL=0
MOVL C00661 V=800.0 PL=0
MOVL C00662 V=800.0 PL=0
MOVL C00663 V=800.0 PL=0
MOVL C00664 V=800.0 PL=0
MOVL C00665 V=800.0 PL=0
MOVL C00666 V=800.0 PL=0
MOVL C00667 V=800.0 PL=0
MOVL C00668 V=800.0 PL=0
MOVL C00669 V=800.0 PL=0
MOVL C00670 V=800.0 PL=0
MOVL C00671 V=800.0 PL=0
MOVL C00672 V=800.0 PL=0
MOVL C00673 V=800.0 PL=0
MOVL C00674 V=800.0 PL=0
MOVL C00675 V=800.0 PL=0
MOVL C00676 V=800.0 PL=0
MOVL C00677 V=800.0 PL=0
MOVL C00678 V=800.0 PL=0
MOVL C00679 V=800.0 PL=0
MOVL C00680 V=800.0 PL=0
MOVL C00681 V=800.0 PL=0
MOVL C00682 V=800.0 PL=0
MOVL C00683 V=800.0 PL=0
MOVL C00684 V=800.0 PL=0
MOVL C00685 V=800.0 PL=0
MOVL C00686 V=800.0 PL=0
MOVL C00687 V=800.0 PL=0
MOVL C00688 V=800.0 PL=0
MOVL C00689 V=800.0 PL=0
MOVL C00690 V=800.0 PL=0
MOVL C00691 V=800.0 PL=0
MOVL C00692 V=800.0 PL=0
MOVL C00693 V=800.0 PL=0
MOVL C00694 V=800.0 PL=0
MOVL C00695 V=800.0 PL=0
MOVL C00696 V=800.0 PL=0
MOVL C00697 V=800.0 PL=0
MOVL C00698 V=800.0 PL=0
MOVL C00699 V=800.0 PL=0
MOVL C00700 V=800.0 PL=0
MOVL C00701 V=800.0 PL=0
MOVL C00702 V=800.0 PL=0
MOVL C00703 V=800.0 PL=0
MOVL C00704 V=800.0 PL=0
MOVL C00705 V=800.0 PL=0
MOVL C00706 V=800.0 PL=0
MOVL C00707 V=800.0 PL=0
MOVL C00708 V=800.0 PL=0
MOVL C00709 V=800.0 PL=0
MOVL C00710 V=800.0 PL=0
MOVL C00711 V=800.0 PL=0
MOVL C00712 V=800.0 PL=0
MOVL C00713 V=800.0 PL=0
MOVL C00714 V=800.0 PL=0
MOVL C00715 V=800.0 PL=0
MOVL C00716 V=800.0 PL=0
MOVL C00717 V=800.0 PL=0
MOVL C00718 V=800.0 PL=0
MOVL C00719 V=800.0 PL=0
MOVL C00720 V=800.0 PL=0
MOVL C00721 V=800.0 PL=0
MOVL C00722 V=800.0 PL=0
MOVL C00723 V=800.0 PL=0
MOVL C00724 V=800.0 PL=0
MOVL C00725 V=800.0 PL=0
MOVL C00726 V=800.0 PL=0
MOVL C00727 V=800.0 PL=0
MOVL C00728 V=800.0 PL=0
MOVL C00729 V=800.0 PL=0
MOVL C00730 V=800.0 PL=0
MOVL C00731 V=800.0 PL=0
MOVL C00732 V=800.0 PL=0
MOVL C00733 V=800.0 PL=0
MOVL C00734 V=800.0 PL=0
MOVL C00735 V=800.0 PL=0
MOVL C00736 V=800.0 PL=0
MOVL C00737 V=800.0 PL=0
MOVL C00738 V=800.0 PL=0
MOVL C00739 V=800.0 PL=0
MOVL C00740 V=800.0 PL=0
MOVL C00741 V=800.0 PL=0
MOVL C00742 V=800.0 PL=0
MOVL C00743 V=800.0 PL=0
MOVL C00744 V=800.0 PL=0
MOVL C00745 V=800.0 PL=0
MOVL C00746 V=800.0 PL=0
MOVL C00747 V=800.0 PL=0
MOVL C00748 V=800.0 PL=0
MOVL C00749 V=800.0 PL=0
MOVL C00750 V=800.0 PL=0
MOVL C00751 V=800.0 PL=0
MOVL C00752 V=800.0 PL=0
MOVL C00753 V=800.0 PL=0
MOVL C00754 V=800.0 PL=0
MOVL C00755 V=800.0 PL=0
MOVL C00756 V=800.0 PL=0
MOVL C00757 V=800.0 PL=0
MOVL C00758 V=800.0 PL=0
MOVL C00759 V=800.0 PL=0
MOVL C00760 V=800.0 PL=0
MOVL C00761 V=800.0 PL=0
MOVL C00762 V=800.0 PL=0
MOVL C00763 V=800.0 PL=0
MOVL C00764 V=800.0 PL=0
MOVL C00765 V=800.0 PL=0
MOVL C00766 V=800.0 PL=0
MOVL C00767 V=800.0 PL=0
MOVL C00768 V=800.0 PL=0
MOVL C00769 V=800.0 PL=0
MOVL C00770 V=800.0 PL=0
MOVL C00771 V=800.0 PL=0
MOVL C00772 V=800.0 PL=0
MOVL C00773 V=800.0 PL=0
MOVL C00774 V=800.0 PL=0
MOVL C00775 V=800.0 PL=0
MOVL C00776 V=800.0 PL=0
MOVL C00777 V=800.0 PL=0
MOVL C00778 V=800.0 PL=0
MOVL C00779 V=800.0 PL=0
MOVL C00780 V=800.0 PL=0
MOVL C00781 V=800.0 PL=0
MOVL C00782 V=800.0 PL=0
MOVL C00783 V=800.0 PL=0
MOVL C00784 V=800.0 PL=0
MOVL C00785 V=800.0 PL=0
MOVL C00786 V=800.0 PL=0
MOVL C00787 V=800.0 PL=0
MOVL C00788 V=800.0 PL=0
MOVL C00789 V=800.0 PL=0
MOVL C00790 V=800.0 PL=0
MOVL C00791 V=800.0 PL=0
MOVL C00792 V=800.0 PL=0
MOVL C00793 V=800.0 PL=0
MOVL C00794 V=800.0 PL=0
MOVL C00795 V=800.0 PL=0
MOVL C00796 V=800.0 PL=0
MOVL C00797 V=800.0 PL=0
MOVL C00798 V=800.0 PL=0
MOVL C00799 V=800.0 PL=0
MOVL C00800 V=800.0 PL=0
MOVL C00801 V=800.0 PL=0
MOVL C00802 V=800.0 PL=0
MOVL C00803 V=800.0 PL=0
MOVL C00804 V=800.0 PL=0
MOVL C00805 V=800.0 PL=0
MOVL C00806 V=800.0 PL=0
MOVL C00807 V=800.0 PL=0
MOVL C00808 V=800.0 PL=0
MOVL C00809 V=800.0 PL=0
MOVL C00810 V=800.0 PL=0
MOVL C00811 V=800.0 PL=0
MOVL C00812 V=800.0 PL=0
MOVL C00813 V=800.0 PL=0
MOVL C00814 V=800.0 PL=0
MOVL C00815 V=800.0 PL=0
MOVL C00816 V=800.0 PL=0
MOVL C00817 V=800.0 PL=0
MOVL C00818 V=800.0 PL=0
MOVL C00819 V=800.0 PL=0
MOVL C00820 V=800.0 PL=0
MOVL C00821 V=800.0 PL=0
MOVL C00822 V=800.0 PL=0
MOVL C00823 V=800.0 PL=0
MOVL C00824 V=800.0 PL=0
MOVL C00825 V=800.0 PL=0
MOVL C00826 V=800.0 PL=0
MOVL C00827 V=800.0 PL=0
MOVL C00828 V=800.0 PL=0
MOVL C00829 V=800.0 PL=0
MOVL C00830 V=800.0 PL=0
MOVL C00831 V=800.0 PL=0
MOVL C00832 V=800.0 PL=0
MOVL C00833 V=800.0 PL=0
MOVL C00834 V=800.0 PL=0
MOVL C00835 V=800.0 PL=0
MOVL C00836 V=800.0 PL=0
MOVL C00837 V=800.0 PL=0
MOVL C00838 V=800.0 PL=0
MOVL C00839 V=800.0 PL=0
MOVL C00840 V=800.0 PL=0
MOVL C00841 V=800.0 PL=0
MOVL C00842 V=800.0 PL=0
MOVL C00843 V=800.0 PL=0
MOVL C00844 V=800.0 PL=0
MOVL C00845 V=800.0 PL=0
MOVL C00846 V=800.0 PL=0
MOVL C00847 V=800.0 PL=0
MOVL C00848 V=800.0 PL=0
MOVL C00849 V=800.0 PL=0
MOVL C00850 V=800.0 PL=0
MOVL C00851 V=800.0 PL=0
MOVL C00852 V=800.0 PL=0
MOVL C00853 V=800.0 PL=0
MOVL C00854 V=800.0 PL=0
MOVL C00855 V=800.0 PL=0
MOVL C00856 V=800.0 PL=0
MOVL C00857 V=800.0 PL=0
MOVL C00858 V=800.0 PL=0
MOVL C00859 V=800.0 PL=0
MOVL C00860 V=800.0 PL=0
MOVL C00861 V=800.0 PL=0
MOVL C00862 V=800.0 PL=0
MOVL C00863 V=800.0 PL=0
MOVL C00864 V=800.0 PL=0
MOVL C00865 V=800.0 PL=0
MOVL C00866 V=800.0 PL=0
MOVL C00867 V=800.0 PL=0
MOVL C00868 V=800.0 PL=0
MOVL C00869 V=800.0 PL=0
MOVL C00870 V=800.0 PL=0
MOVL C00871 V=800.0 PL=0
MOVL C00872 V=800.0 PL=0
MOVL C00873 V=800.0 PL=0
MOVL C00874 V=800.0 PL=0
MOVL C00875 V=800.0 PL=0
MOVL C00876 V=800.0 PL=0
MOVL C00877 V=800.0 PL=0
MOVL C00878 V=800.0 PL=0
MOVL C00879 V=800.0 PL=0
MOVL C00880 V=800.0 PL=0
MOVL C00881 V=800.0 PL=0
MOVL C00882 V=800.0 PL=0
MOVL C00883 V=800.0 PL=0
MOVL C00884 V=800.0 PL=0
MOVL C00885 V=800.0 PL=0
MOVL C00886 V=800.0 PL=0
MOVL C00887 V=800.0 PL=0
MOVL C00888 V=800.0 PL=0
MOVL C00889 V=800.0 PL=0
MOVL C00890 V=800.0 PL=0
MOVL C00891 V=800.0 PL=0
MOVL C00892 V=800.0 PL=0
MOVL C00893 V=800.0 PL=0
MOVL C00894 V=800.0 PL=0
MOVL C00895 V=800.0 PL=0
MOVL C00896 V=800.0 PL=0
MOVL C00897 V=800.0 PL=0
MOVL C00898 V=800.0 PL=0
MOVL C00899 V=800.0 PL=0
MOVL C00900 V=800.0 PL=0
MOVL C00901 V=800.0 PL=0
MOVL C00902 V=800.0 PL=0
MOVL C00903 V=800.0 PL=0
MOVL C00904 V=800.0 PL=0
MOVL C00905 V=800.0 PL=0
MOVL C00906 V=800.0 PL=0
MOVL C00907 V=800.0 PL=0
MOVL C00908 V=800.0 PL=0
MOVL C00909 V=800.0 PL=0
MOVL C00910 V=800.0 PL=0
MOVL C00911 V=800.0 PL=0
MOVL C00912 V=800.0 PL=0
MOVL C00913 V=800.0 PL=0
MOVL C00914 V=800.0 PL=0
MOVL C00915 V=800.0 PL=0
MOVL C00916 V=800.0 PL=0
MOVL C00917 V=800.0 PL=0
MOVL C00918 V=800.0 PL=0
MOVL C00919 V=800.0 PL=0
MOVL C00920 V=800.0 PL=0
MOVL C00921 V=800.0 PL=0
MOVL C00922 V=800.0 PL=0
MOVL C00923 V=800.0 PL=0
MOVL C00924 V=800.0 PL=0
MOVL C00925 V=800.0 PL=0
MOVL C00926 V=800.0 PL=0
MOVL C00927 V=800.0 PL=0
MOVL C00928 V=800.0 PL=0
MOVL C00929 V=800.0 PL=0
MOVL C00930 V=800.0 PL=0
MOVL C00931 V=800.0 PL=0
MOVL C00932 V=800.0 PL=0
MOVL C00933 V=800.0 PL=0
MOVL C00934 V=800.0 PL=0
MOVL C00935 V=800.0 PL=0
MOVL C00936 V=800.0 PL=0
MOVL C00937 V=800.0 PL=0
MOVL C00938 V=800.0 PL=0
MOVL C00939 V=800.0 PL=0
MOVL C00940 V=800.0 PL=0
MOVL C00941 V=800.0 PL=0
MOVL C00942 V=800.0 PL=0
MOVL C00943 V=800.0 PL=0
MOVL C00944 V=800.0 PL=0
MOVL C00945 V=800.0 PL=0
MOVL C00946 V=800.0 PL=0
MOVL C00947 V=800.0 PL=0
MOVL C00948 V=800.0 PL=0
MOVL C00949 V=800.0 PL=0
MOVL C00950 V=800.0 PL=0
MOVL C00951 V=800.0 PL=0
MOVL C00952 V=800.0 PL=0
MOVL C00953 V=800.0 PL=0
MOVL C00954 V=800.0 PL=0
MOVL C00955 V=800.0 PL=0
MOVL C00956 V=800.0 PL=0
MOVL C00957 V=800.0 PL=0
MOVL C00958 V=800.0 PL=0
MOVL C00959 V=800.0 PL=0
MOVL C00960 V=800.0 PL=0
MOVL C00961 V=800.0 PL=0
MOVL C00962 V=800.0 PL=0
MOVL C00963 V=800.0 PL=0
MOVL C00964 V=800.0 PL=0
MOVL C00965 V=800.0 PL=0
MOVL C00966 V=800.0 PL=0
MOVL C00967 V=800.0 PL=0
MOVL C00968 V=800.0 PL=0
MOVL C00969 V=800.0 PL=0
MOVL C00970 V=800.0 PL=0
MOVL C00971 V=800.0 PL=0
MOVL C00972 V=800.0 PL=0
MOVL C00973 V=800.0 PL=0
MOVL C00974 V=800.0 PL=0
MOVL C00975 V=800.0 PL=0
MOVL C00976 V=800.0 PL=0
MOVL C00977 V=800.0 PL=0
MOVL C00978 V=800.0 PL=0
MOVL C00979 V=800.0 PL=0
MOVL C00980 V=800.0 PL=0
MOVL C00981 V=800.0 PL=0
MOVL C00982 V=800.0 PL=0
MOVL C00983 V=800.0 PL=0
MOVL C00984 V=800.0 PL=0
MOVL C00985 V=800.0 PL=0
MOVL C00986 V=800.0 PL=0
MOVL C00987 V=800.0 PL=0
MOVL C00988 V=800.0 PL=0
MOVL C00989 V=800.0 PL=0
MOVL C00990 V=800.0 PL=0
MOVL C00991 V=800.0 PL=0
MOVL C00992 V=800.0 PL=0
MOVL C00993 V=800.0 PL=0
MOVL C00994 V=800.0 PL=0
MOVL C00995 V=800.0 PL=0
MOVL C00996 V=800.0 PL=0
MOVL C00997 V=800.0 PL=0
MOVL C00998 V=800.0 PL=0
MOVL C00999 V=800.0 PL=0
MOVL C01000 V=800.0 PL=0
MOVL C01001 V=800.0 PL=0
MOVL C01002 V=800.0 PL=0
MOVL C01003 V=800.0 PL=0
MOVL C01004 V=800.0 PL=0
MOVL C01005 V=800.0 PL=0
MOVL C01006 V=800.0 PL=0
MOVL C01007 V=800.0 PL=0
MOVL C01008 V=800.0 PL=0
MOVL C01009 V=800.0 PL=0
MOVL C01010 V=800.0 PL=0
MOVL C01011 V=800.0 PL=0
MOVL C01012 V=800.0 PL=0
MOVL C01013 V=800.0 PL=0
MOVL C01014 V=800.0 PL=0
MOVL C01015 V=800.0 PL=0
MOVL C01016 V=800.0 PL=0
MOVL C01017 V=800.0 PL=0
MOVL C01018 V=800.0 PL=0
MOVL C01019 V=800.0 PL=0
MOVL C01020 V=800.0 PL=0
MOVL C01021 V=800.0 PL=0
MOVL C01022 V=800.0 PL=0
MOVL C01023 V=800.0 PL=0
MOVL C01024 V=800.0 PL=0
MOVL C01025 V=800.0 PL=0
MOVL C01026 V=800.0 PL=0
MOVL C01027 V=800.0 PL=0
MOVL C01028 V=800.0 PL=0
MOVL C01029 V=800.0 PL=0
MOVL C01030 V=800.0 PL=0
MOVL C01031 V=800.0 PL=0
MOVL C01032 V=800.0 PL=0
MOVL C01033 V=800.0 PL=0
MOVL C01034 V=800.0 PL=0
MOVL C01035 V=800.0 PL=0
MOVL C01036 V=800.0 PL=0
MOVL C01037 V=800.0 PL=0
MOVL C01038 V=800.0 PL=0
MOVL C01039 V=800.0 PL=0
MOVL C01040 V=800.0 PL=0
MOVL C01041 V=800.0 PL=0
MOVL C01042 V=800.0 PL=0
MOVL C01043 V=800.0 PL=0
MOVL C01044 V=800.0 PL=0
MOVL C01045 V=800.0 PL=0
MOVL C01046 V=800.0 PL=0
MOVL C01047 V=800.0 PL=0
MOVL C01048 V=800.0 PL=0
MOVL C01049 V=800.0 PL=0
MOVL C01050 V=800.0 PL=0
MOVL C01051 V=800.0 PL=0
MOVL C01052 V=800.0 PL=0
MOVL C01053 V=800.0 PL=0
MOVL C01054 V=800.0 PL=0
MOVL C01055 V=800.0 PL=0
MOVL C01056 V=800.0 PL=0
MOVL C01057 V=800.0 PL=0
MOVL C01058 V=800.0 PL=0
MOVL C01059 V=800.0 PL=0
MOVL C01060 V=800.0 PL=0
MOVL C01061 V=800.0 PL=0
MOVL C01062 V=800.0 PL=0
MOVL C01063 V=800.0 PL=0
MOVL C01064 V=800.0 PL=0
MOVL C01065 V=800.0 PL=0
MOVL C01066 V=800.0 PL=0
MOVL C01067 V=800.0 PL=0
MOVL C01068 V=800.0 PL=0
MOVL C01069 V=800.0 PL=0
MOVL C01070 V=800.0 PL=0
MOVL C01071 V=800.0 PL=0
MOVL C01072 V=800.0 PL=0
MOVL C01073 V=800.0 PL=0
MOVL C01074 V=800.0 PL=0
MOVL C01075 V=800.0 PL=0
MOVL C01076 V=800.0 PL=0
MOVL C01077 V=800.0 PL=0
MOVL C01078 V=800.0 PL=0
MOVL C01079 V=800.0 PL=0
MOVL C01080 V=800.0 PL=0
MOVL C01081 V=800.0 PL=0
MOVL C01082 V=800.0 PL=0
MOVL C01083 V=800.0 PL=0
MOVL C01084 V=800.0 PL=0
MOVL C01085 V=800.0 PL=0
MOVL C01086 V=800.0 PL=0
MOVL C01087 V=800.0 PL=0
MOVL C01088 V=800.0 PL=0
MOVL C01089 V=800.0 PL=0
MOVL C01090 V=800.0 PL=0
MOVL C01091 V=800.0 PL=0
MOVL C01092 V=800.0 PL=0
MOVL C01093 V=800.0 PL=0
MOVL C01094 V=800.0 PL=0
MOVL C01095 V=800.0 PL=0
MOVL C01096 V=800.0 PL=0
MOVL C01097 V=800.0 PL=0
MOVL C01098 V=800.0 PL=0
MOVL C01099 V=800.0 PL=0
MOVL C01100 V=800.0 PL=0
MOVL C01101 V=800.0 PL=0
MOVL C01102 V=800.0 PL=0
MOVL C01103 V=800.0 PL=0
MOVL C01104 V=800.0 PL=0
MOVL C01105 V=800.0 PL=0
MOVL C01106 V=800.0 PL=0
MOVL C01107 V=800.0 PL=0
MOVL C01108 V=800.0 PL=0
MOVL C01109 V=800.0 PL=0
MOVL C01110 V=800.0 PL=0
MOVL C01111 V=800.0 PL=0
MOVL C01112 V=800.0 PL=0
MOVL C01113 V=800.0 PL=0
MOVL C01114 V=800.0 PL=0
MOVL C01115 V=800.0 PL=0
MOVL C01116 V=800.0 PL=0
MOVL C01117 V=800.0 PL=0
MOVL C01118 V=800.0 PL=0
MOVL C01119 V=800.0 PL=0
MOVL C01120 V=800.0 PL=0
MOVL C01121 V=800.0 PL=0
MOVL C01122 V=800.0 PL=0
MOVL C01123 V=800.0 PL=0
MOVL C01124 V=800.0 PL=0
MOVL C01125 V=800.0 PL=0
MOVL C01126 V=800.0 PL=0
MOVL C01127 V=800.0 PL=0
MOVL C01128 V=800.0 PL=0
MOVL C01129 V=800.0 PL=0
MOVL C01130 V=800.0 PL=0
MOVL C01131 V=800.0 PL=0
MOVL C01132 V=800.0 PL=0
MOVL C01133 V=800.0 PL=0
MOVL C01134 V=800.0 PL=0
MOVL C01135 V=800.0 PL=0
MOVL C01136 V=800.0 PL=0
MOVL C01137 V=800.0 PL=0
MOVL C01138 V=800.0 PL=0
MOVL C01139 V=800.0 PL=0
MOVL C01140 V=800.0 PL=0
MOVL C01141 V=800.0 PL=0
MOVL C01142 V=800.0 PL=0
MOVL C01143 V=800.0 PL=0
MOVL C01144 V=800.0 PL=0
MOVL C01145 V=800.0 PL=0
MOVL C01146 V=800.0 PL=0
MOVL C01147 V=800.0 PL=0
MOVL C01148 V=800.0 PL=0
MOVL C01149 V=800.0 PL=0
MOVL C01150 V=800.0 PL=0
MOVL C01151 V=800.0 PL=0
MOVL C01152 V=800.0 PL=0
MOVL C01153 V=800.0 PL=0
MOVL C01154 V=800.0 PL=0
MOVL C01155 V=800.0 PL=0
MOVL C01156 V=800.0 PL=0
MOVL C01157 V=800.0 PL=0
MOVL C01158 V=800.0 PL=0
MOVL C01159 V=800.0 PL=0
MOVL C01160 V=800.0 PL=0
MOVL C01161 V=800.0 PL=0
MOVL C01162 V=800.0 PL=0
MOVL C01163 V=800.0 PL=0
MOVL C01164 V=800.0 PL=0
MOVL C01165 V=800.0 PL=0
MOVL C01166 V=800.0 PL=0
MOVL C01167 V=800.0 PL=0
MOVL C01168 V=800.0 PL=0
MOVL C01169 V=800.0 PL=0
MOVL C01170 V=800.0 PL=0
MOVL C01171 V=800.0 PL=0
MOVL C01172 V=800.0 PL=0
MOVL C01173 V=800.0 PL=0
MOVL C01174 V=800.0 PL=0
MOVL C01175 V=800.0 PL=0
MOVL C01176 V=800.0 PL=0
MOVL C01177 V=800.0 PL=0
MOVL C01178 V=800.0 PL=0
MOVL C01179 V=800.0 PL=0
MOVL C01180 V=800.0 PL=0
MOVL C01181 V=800.0 PL=0
MOVL C01182 V=800.0 PL=0
MOVL C01183 V=800.0 PL=0
MOVL C01184 V=800.0 PL=0
MOVL C01185 V=800.0 PL=0
MOVL C01186 V=800.0 PL=0
MOVL C01187 V=800.0 PL=0
MOVL C01188 V=800.0 PL=0
MOVL C01189 V=800.0 PL=0
MOVL C01190 V=800.0 PL=0
MOVL C01191 V=800.0 PL=0
MOVL C01192 V=800.0 PL=0
MOVL C01193 V=800.0 PL=0
MOVL C01194 V=800.0 PL=0
MOVL C01195 V=800.0 PL=0
MOVL C01196 V=800.0 PL=0
MOVL C01197 V=800.0 PL=0
MOVL C01198 V=800.0 PL=0
MOVL C01199 V=800.0 PL=0
MOVL C01200 V=800.0 PL=0
MOVL C01201 V=800.0 PL=0
MOVL C01202 V=800.0 PL=0
MOVL C01203 V=800.0 PL=0
MOVL C01204 V=800.0 PL=0
MOVL C01205 V=800.0 PL=0
MOVL C01206 V=800.0 PL=0
MOVL C01207 V=800.0 PL=0
MOVL C01208 V=800.0 PL=0
MOVL C01209 V=800.0 PL=0
MOVL C01210 V=800.0 PL=0
MOVL C01211 V=800.0 PL=0
MOVL C01212 V=800.0 PL=0
MOVL C01213 V=800.0 PL=0
MOVL C01214 V=800.0 PL=0
MOVL C01215 V=800.0 PL=0
MOVL C01216 V=800.0 PL=0
MOVL C01217 V=800.0 PL=0
MOVL C01218 V=800.0 PL=0
MOVL C01219 V=800.0 PL=0
MOVL C01220 V=800.0 PL=0
MOVL C01221 V=800.0 PL=0
MOVL C01222 V=800.0 PL=0
MOVL C01223 V=800.0 PL=0
MOVL C01224 V=800.0 PL=0
MOVL C01225 V=800.0 PL=0
MOVL C01226 V=800.0 PL=0
MOVL C01227 V=800.0 PL=0
MOVL C01228 V=800.0 PL=0
MOVL C01229 V=800.0 PL=0
MOVL C01230 V=800.0 PL=0
MOVL C01231 V=800.0 PL=0
MOVL C01232 V=800.0 PL=0
MOVL C01233 V=800.0 PL=0
MOVL C01234 V=800.0 PL=0
MOVL C01235 V=800.0 PL=0
MOVL C01236 V=800.0 PL=0
MOVL C01237 V=800.0 PL=0
MOVL C01238 V=800.0 PL=0
MOVL C01239 V=800.0 PL=0
MOVL C01240 V=800.0 PL=0
MOVL C01241 V=800.0 PL=0
MOVL C01242 V=800.0 PL=0
MOVL C01243 V=800.0 PL=0
MOVL C01244 V=800.0 PL=0
MOVL C01245 V=800.0 PL=0
MOVL C01246 V=800.0 PL=0
MOVL C01247 V=800.0 PL=0
MOVL C01248 V=800.0 PL=0
MOVL C01249 V=800.0 PL=0
MOVL C01250 V=800.0 PL=0
MOVL C01251 V=800.0 PL=0
MOVL C01252 V=800.0 PL=0
MOVL C01253 V=800.0 PL=0
MOVL C01254 V=800.0 PL=0
MOVL C01255 V=800.0 PL=0
MOVL C01256 V=800.0 PL=0
MOVL C01257 V=800.0 PL=0
MOVL C01258 V=800.0 PL=0
MOVL C01259 V=800.0 PL=0
MOVL C01260 V=800.0 PL=0
MOVL C01261 V=800.0 PL=0
MOVL C01262 V=800.0 PL=0
MOVL C01263 V=800.0 PL=0
MOVL C01264 V=800.0 PL=0
MOVL C01265 V=800.0 PL=0
MOVL C01266 V=800.0 PL=0
MOVL C01267 V=800.0 PL=0
MOVL C01268 V=800.0 PL=0
MOVL C01269 V=800.0 PL=0
MOVL C01270 V=800.0 PL=0
MOVL C01271 V=800.0 PL=0
MOVL C01272 V=800.0 PL=0
MOVL C01273 V=800.0 PL=0
MOVL C01274 V=800.0 PL=0
MOVL C01275 V=800.0 PL=0
MOVL C01276 V=800.0 PL=0
MOVL C01277 V=800.0 PL=0
MOVL C01278 V=800.0 PL=0
MOVL C01279 V=800.0 PL=0
MOVL C01280 V=800.0 PL=0
MOVL C01281 V=800.0 PL=0
MOVL C01282 V=800.0 PL=0
MOVL C01283 V=800.0 PL=0
MOVL C01284 V=800.0 PL=0
MOVL C01285 V=800.0 PL=0
MOVL C01286 V=800.0 PL=0
MOVL C01287 V=800.0 PL=0
MOVL C01288 V=800.0 PL=0
MOVL C01289 V=800.0 PL=0
MOVL C01290 V=800.0 PL=0
MOVL C01291 V=800.0 PL=0
MOVL C01292 V=800.0 PL=0
MOVL C01293 V=800.0 PL=0
MOVL C01294 V=800.0 PL=0
MOVL C01295 V=800.0 PL=0
MOVL C01296 V=800.0 PL=0
MOVL C01297 V=800.0 PL=0
MOVL C01298 V=800.0 PL=0
MOVL C01299 V=800.0 PL=0
MOVL C01300 V=800.0 PL=0
MOVL C01301 V=800.0 PL=0
MOVL C01302 V=800.0 PL=0
MOVL C01303 V=800.0 PL=0
MOVL C01304 V=800.0 PL=0
MOVL C01305 V=800.0 PL=0
MOVL C01306 V=800.0 PL=0
MOVL C01307 V=800.0 PL=0
MOVL C01308 V=800.0 PL=0
MOVL C01309 V=800.0 PL=0
MOVL C01310 V=800.0 PL=0
MOVL C01311 V=800.0 PL=0
MOVL C01312 V=800.0 PL=0
MOVL C01313 V=800.0 PL=0
MOVL C01314 V=800.0 PL=0
MOVL C01315 V=800.0 PL=0
MOVL C01316 V=800.0 PL=0
MOVL C01317 V=800.0 PL=0
MOVL C01318 V=800.0 PL=0
MOVL C01319 V=800.0 PL=0
MOVL C01320 V=800.0 PL=0
MOVL C01321 V=800.0 PL=0
MOVL C01322 V=800.0 PL=0
MOVL C01323 V=800.0 PL=0
MOVL C01324 V=800.0 PL=0
MOVL C01325 V=800.0 PL=0
MOVL C01326 V=800.0 PL=0
MOVL C01327 V=800.0 PL=0
MOVL C01328 V=800.0 PL=0
MOVL C01329 V=800.0 PL=0
MOVL C01330 V=800.0 PL=0
MOVL C01331 V=800.0 PL=0
MOVL C01332 V=800.0 PL=0
MOVL C01333 V=800.0 PL=0
MOVL C01334 V=800.0 PL=0
MOVL C01335 V=800.0 PL=0
MOVL C01336 V=800.0 PL=0
MOVL C01337 V=800.0 PL=0
MOVL C01338 V=800.0 PL=0
MOVL C01339 V=800.0 PL=0
MOVL C01340 V=800.0 PL=0
MOVL C01341 V=800.0 PL=0
MOVL C01342 V=800.0 PL=0
MOVL C01343 V=800.0 PL=0
MOVL C01344 V=800.0 PL=0
MOVL C01345 V=800.0 PL=0
MOVL C01346 V=800.0 PL=0
MOVL C01347 V=800.0 PL=0
MOVL C01348 V=800.0 PL=0
MOVL C01349 V=800.0 PL=0
MOVL C01350 V=800.0 PL=0
MOVL C01351 V=800.0 PL=0
MOVL C01352 V=800.0 PL=0
MOVL C01353 V=800.0 PL=0
MOVL C01354 V=800.0 PL=0
MOVL C01355 V=800.0 PL=0
MOVL C01356 V=800.0 PL=0
MOVL C01357 V=800.0 PL=0
MOVL C01358 V=800.0 PL=0
MOVL C01359 V=800.0 PL=0
MOVL C01360 V=800.0 PL=0
MOVL C01361 V=800.0 PL=0
MOVL C01362 V=800.0 PL=0
MOVL C01363 V=800.0 PL=0
MOVL C01364 V=800.0 PL=0
MOVL C01365 V=800.0 PL=0
MOVL C01366 V=800.0 PL=0
MOVL C01367 V=800.0 PL=0
MOVL C01368 V=800.0 PL=0
MOVL C01369 V=800.0 PL=0
MOVL C01370 V=800.0 PL=0
MOVL C01371 V=800.0 PL=0
MOVL C01372 V=800.0 PL=0
MOVL C01373 V=800.0 PL=0
MOVL C01374 V=800.0 PL=0
MOVL C01375 V=800.0 PL=0
MOVL C01376 V=800.0 PL=0
MOVL C01377 V=800.0 PL=0
MOVL C01378 V=800.0 PL=0
MOVL C01379 V=800.0 PL=0
MOVL C01380 V=800.0 PL=0
MOVL C01381 V=800.0 PL=0
MOVL C01382 V=800.0 PL=0
MOVL C01383 V=800.0 PL=0
MOVL C01384 V=800.0 PL=0
MOVL C01385 V=800.0 PL=0
MOVL C01386 V=800.0 PL=0
MOVL C01387 V=800.0 PL=0
MOVL C01388 V=800.0 PL=0
MOVL C01389 V=800.0 PL=0
MOVL C01390 V=800.0 PL=0
MOVL C01391 V=800.0 PL=0
MOVL C01392 V=800.0 PL=0
MOVL C01393 V=800.0 PL=0
MOVL C01394 V=800.0 PL=0
MOVL C01395 V=800.0 PL=0
MOVL C01396 V=800.0 PL=0
MOVL C01397 V=800.0 PL=0
MOVL C01398 V=800.0 PL=0
MOVL C01399 V=800.0 PL=0
MOVL C01400 V=800.0 PL=0
MOVL C01401 V=800.0 PL=0
MOVL C01402 V=800.0 PL=0
MOVL C01403 V=800.0 PL=0
MOVL C01404 V=800.0 PL=0
MOVL C01405 V=800.0 PL=0
MOVL C01406 V=800.0 PL=0
MOVL C01407 V=800.0 PL=0
MOVL C01408 V=800.0 PL=0
MOVL C01409 V=800.0 PL=0
MOVL C01410 V=800.0 PL=0
MOVL C01411 V=800.0 PL=0
MOVL C01412 V=800.0 PL=0
MOVL C01413 V=800.0 PL=0
MOVL C01414 V=800.0 PL=0
MOVL C01415 V=800.0 PL=0
MOVL C01416 V=800.0 PL=0
MOVL C01417 V=800.0 PL=0
MOVL C01418 V=800.0 PL=0
MOVL C01419 V=800.0 PL=0
MOVL C01420 V=800.0 PL=0
MOVL C01421 V=800.0 PL=0
MOVL C01422 V=800.0 PL=0
MOVL C01423 V=800.0 PL=0
MOVL C01424 V=800.0 PL=0
MOVL C01425 V=800.0 PL=0
MOVL C01426 V=800.0 PL=0
MOVL C01427 V=800.0 PL=0
MOVL C01428 V=800.0 PL=0
MOVL C01429 V=800.0 PL=0
MOVL C01430 V=800.0 PL=0
MOVL C01431 V=800.0 PL=0
MOVL C01432 V=800.0 PL=0
MOVL C01433 V=800.0 PL=0
MOVL C01434 V=800.0 PL=0
MOVL C01435 V=800.0 PL=0
MOVL C01436 V=800.0 PL=0
MOVL C01437 V=800.0 PL=0
MOVL C01438 V=800.0 PL=0
MOVL C01439 V=800.0 PL=0
MOVL C01440 V=800.0 PL=0
MOVL C01441 V=800.0 PL=0
MOVL C01442 V=800.0 PL=0
MOVL C01443 V=800.0 PL=0
MOVL C01444 V=800.0 PL=0
MOVL C01445 V=800.0 PL=0
MOVL C01446 V=800.0 PL=0
MOVL C01447 V=800.0 PL=0
MOVL C01448 V=800.0 PL=0
MOVL C01449 V=800.0 PL=0
MOVL C01450 V=800.0 PL=0
MOVL C01451 V=800.0 PL=0
MOVL C01452 V=800.0 PL=0
MOVL C01453 V=800.0 PL=0
MOVL C01454 V=800.0 PL=0
MOVL C01455 V=800.0 PL=0
MOVL C01456 V=800.0 PL=0
MOVL C01457 V=800.0 PL=0
MOVL C01458 V=800.0 PL=0
MOVL C01459 V=800.0 PL=0
MOVL C01460 V=800.0 PL=0
MOVL C01461 V=800.0 PL=0
MOVL C01462 V=800.0 PL=0
MOVL C01463 V=800.0 PL=0
MOVL C01464 V=800.0 PL=0
MOVL C01465 V=800.0 PL=0
MOVL C01466 V=800.0 PL=0
MOVL C01467 V=800.0 PL=0
MOVL C01468 V=800.0 PL=0
MOVL C01469 V=800.0 PL=0
MOVL C01470 V=800.0 PL=0
MOVL C01471 V=800.0 PL=0
MOVL C01472 V=800.0 PL=0
MOVL C01473 V=800.0 PL=0
MOVL C01474 V=800.0 PL=0
MOVL C01475 V=800.0 PL=0
MOVL C01476 V=800.0 PL=0
MOVL C01477 V=800.0 PL=0
MOVL C01478 V=800.0 PL=0
MOVL C01479 V=800.0 PL=0
MOVL C01480 V=800.0 PL=0
MOVL C01481 V=800.0 PL=0
MOVL C01482 V=800.0 PL=0
MOVL C01483 V=800.0 PL=0
MOVL C01484 V=800.0 PL=0
MOVL C01485 V=800.0 PL=0
MOVL C01486 V=800.0 PL=0
MOVL C01487 V=800.0 PL=0
MOVL C01488 V=800.0 PL=0
MOVL C01489 V=800.0 PL=0
MOVL C01490 V=800.0 PL=0
MOVL C01491 V=800.0 PL=0
MOVL C01492 V=800.0 PL=0
MOVL C01493 V=800.0 PL=0
MOVL C01494 V=800.0 PL=0
MOVL C01495 V=800.0 PL=0
MOVL C01496 V=800.0 PL=0
MOVL C01497 V=800.0 PL=0
MOVL C01498 V=800.0 PL=0
MOVL C01499 V=800.0 PL=0
MOVL C01500 V=800.0 PL=0
MOVL C01501 V=800.0 PL=0
MOVL C01502 V=800.0 PL=0
MOVL C01503 V=800.0 PL=0
MOVL C01504 V=800.0 PL=0
MOVL C01505 V=800.0 PL=0
MOVL C01506 V=800.0 PL=0
MOVL C01507 V=800.0 PL=0
MOVL C01508 V=800.0 PL=0
MOVL C01509 V=800.0 PL=0
MOVL C01510 V=800.0 PL=0
MOVL C01511 V=800.0 PL=0
MOVL C01512 V=800.0 PL=0
MOVL C01513 V=800.0 PL=0
MOVL C01514 V=800.0 PL=0
MOVL C01515 V=800.0 PL=0
MOVL C01516 V=800.0 PL=0
MOVL C01517 V=800.0 PL=0
MOVL C01518 V=800.0 PL=0
MOVL C01519 V=800.0 PL=0
MOVL C01520 V=800.0 PL=0
MOVL C01521 V=800.0 PL=0
MOVL C01522 V=800.0 PL=0
MOVL C01523 V=800.0 PL=0
MOVL C01524 V=800.0 PL=0
MOVL C01525 V=800.0 PL=0
MOVL C01526 V=800.0 PL=0
MOVL C01527 V=800.0 PL=0
MOVL C01528 V=800.0 PL=0
MOVL C01529 V=800.0 PL=0
MOVL C01530 V=800.0 PL=0
MOVL C01531 V=800.0 PL=0
MOVL C01532 V=800.0 PL=0
MOVL C01533 V=800.0 PL=0
MOVL C01534 V=800.0 PL=0
MOVL C01535 V=800.0 PL=0
MOVL C01536 V=800.0 PL=0
MOVL C01537 V=800.0 PL=0
MOVL C01538 V=800.0 PL=0
MOVL C01539 V=800.0 PL=0
MOVL C01540 V=800.0 PL=0
MOVL C01541 V=800.0 PL=0
MOVL C01542 V=800.0 PL=0
MOVL C01543 V=800.0 PL=0
MOVL C01544 V=800.0 PL=0
MOVL C01545 V=800.0 PL=0
MOVL C01546 V=800.0 PL=0
MOVL C01547 V=800.0 PL=0
MOVL C01548 V=800.0 PL=0
MOVL C01549 V=800.0 PL=0
MOVL C01550 V=800.0 PL=0
MOVL C01551 V=800.0 PL=0
MOVL C01552 V=800.0 PL=0
MOVL C01553 V=800.0 PL=0
MOVL C01554 V=800.0 PL=0
MOVL C01555 V=800.0 PL=0
MOVL C01556 V=800.0 PL=0
MOVL C01557 V=800.0 PL=0
MOVL C01558 V=800.0 PL=0
MOVL C01559 V=800.0 PL=0
MOVL C01560 V=800.0 PL=0
MOVL C01561 V=800.0 PL=0
MOVL C01562 V=800.0 PL=0
MOVL C01563 V=800.0 PL=0
MOVL C01564 V=800.0 PL=0
MOVL C01565 V=800.0 PL=0
MOVL C01566 V=800.0 PL=0
MOVL C01567 V=800.0 PL=0
MOVL C01568 V=800.0 PL=0
MOVL C01569 V=800.0 PL=0
MOVL C01570 V=800.0 PL=0
MOVL C01571 V=800.0 PL=0
MOVL C01572 V=800.0 PL=0
MOVL C01573 V=800.0 PL=0
MOVL C01574 V=800.0 PL=0
MOVL C01575 V=800.0 PL=0
MOVL C01576 V=800.0 PL=0
MOVL C01577 V=800.0 PL=0
MOVL C01578 V=800.0 PL=0
MOVL C01579 V=800.0 PL=0
MOVL C01580 V=800.0 PL=0
MOVL C01581 V=800.0 PL=0
MOVL C01582 V=800.0 PL=0
MOVL C01583 V=800.0 PL=0
MOVL C01584 V=800.0 PL=0
MOVL C01585 V=800.0 PL=0
MOVL C01586 V=800.0 PL=0
MOVL C01587 V=800.0 PL=0
MOVL C01588 V=800.0 PL=0
MOVL C01589 V=800.0 PL=0
MOVL C01590 V=800.0 PL=0
MOVL C01591 V=800.0 PL=0
MOVL C01592 V=800.0 PL=0
MOVL C01593 V=800.0 PL=0
MOVL C01594 V=800.0 PL=0
MOVL C01595 V=800.0 PL=0
MOVL C01596 V=800.0 PL=0
MOVL C01597 V=800.0 PL=0
MOVL C01598 V=800.0 PL=0
MOVL C01599 V=800.0 PL=0
MOVL C01600 V=800.0 PL=0
MOVL C01601 V=800.0 PL=0
MOVL C01602 V=800.0 PL=0
MOVL C01603 V=800.0 PL=0
MOVL C01604 V=800.0 PL=0
MOVL C01605 V=800.0 PL=0
MOVL C01606 V=800.0 PL=0
MOVL C01607 V=800.0 PL=0
MOVL C01608 V=800.0 PL=0
MOVL C01609 V=800.0 PL=0
MOVL C01610 V=800.0 PL=0
MOVL C01611 V=800.0 PL=0
MOVL C01612 V=800.0 PL=0
MOVL C01613 V=800.0 PL=0
MOVL C01614 V=800.0 PL=0
MOVL C01615 V=800.0 PL=0
MOVL C01616 V=800.0 PL=0
MOVL C01617 V=800.0 PL=0
MOVL C01618 V=800.0 PL=0
MOVL C01619 V=800.0 PL=0
MOVL C01620 V=800.0 PL=0
MOVL C01621 V=800.0 PL=0
MOVL C01622 V=800.0 PL=0
MOVL C01623 V=800.0 PL=0
MOVL C01624 V=800.0 PL=0
MOVL C01625 V=800.0 PL=0
MOVL C01626 V=800.0 PL=0
MOVL C01627 V=800.0 PL=0
MOVL C01628 V=800.0 PL=0
MOVL C01629 V=800.0 PL=0
MOVL C01630 V=800.0 PL=0
MOVL C01631 V=800.0 PL=0
MOVL C01632 V=800.0 PL=0
MOVL C01633 V=800.0 PL=0
MOVL C01634 V=800.0 PL=0
MOVL C01635 V=800.0 PL=0
MOVL C01636 V=800.0 PL=0
MOVL C01637 V=800.0 PL=0
MOVL C01638 V=800.0 PL=0
MOVL C01639 V=800.0 PL=0
MOVL C01640 V=800.0 PL=0
MOVL C01641 V=800.0 PL=0
MOVL C01642 V=800.0 PL=0
MOVL C01643 V=800.0 PL=0
MOVL C01644 V=800.0 PL=0
MOVL C01645 V=800.0 PL=0
MOVL C01646 V=800.0 PL=0
MOVL C01647 V=800.0 PL=0
MOVL C01648 V=800.0 PL=0
MOVL C01649 V=800.0 PL=0
MOVL C01650 V=800.0 PL=0
MOVL C01651 V=800.0 PL=0
MOVL C01652 V=800.0 PL=0
MOVL C01653 V=800.0 PL=0
MOVL C01654 V=800.0 PL=0
MOVL C01655 V=800.0 PL=0
MOVL C01656 V=800.0 PL=0
MOVL C01657 V=800.0 PL=0
MOVL C01658 V=800.0 PL=0
MOVL C01659 V=800.0 PL=0
MOVL C01660 V=800.0 PL=0
MOVL C01661 V=800.0 PL=0
MOVL C01662 V=800.0 PL=0
MOVL C01663 V=800.0 PL=0
MOVL C01664 V=800.0 PL=0
MOVL C01665 V=800.0 PL=0
MOVL C01666 V=800.0 PL=0
MOVL C01667 V=800.0 PL=0
MOVL C01668 V=800.0 PL=0
MOVL C01669 V=800.0 PL=0
MOVL C01670 V=800.0 PL=0
MOVL C01671 V=800.0 PL=0
MOVL C01672 V=800.0 PL=0
MOVL C01673 V=800.0 PL=0
MOVL C01674 V=800.0 PL=0
MOVL C01675 V=800.0 PL=0
MOVL C01676 V=800.0 PL=0
MOVL C01677 V=800.0 PL=0
MOVL C01678 V=800.0 PL=0
MOVL C01679 V=800.0 PL=0
MOVL C01680 V=800.0 PL=0
MOVL C01681 V=800.0 PL=0
MOVL C01682 V=800.0 PL=0
MOVL C01683 V=800.0 PL=0
MOVL C01684 V=800.0 PL=0
MOVL C01685 V=800.0 PL=0
MOVL C01686 V=800.0 PL=0
MOVL C01687 V=800.0 PL=0
MOVL C01688 V=800.0 PL=0
MOVL C01689 V=800.0 PL=0
MOVL C01690 V=800.0 PL=0
MOVL C01691 V=800.0 PL=0
MOVL C01692 V=800.0 PL=0
MOVL C01693 V=800.0 PL=0
MOVL C01694 V=800.0 PL=0
MOVL C01695 V=800.0 PL=0
MOVL C01696 V=800.0 PL=0
MOVL C01697 V=800.0 PL=0
MOVL C01698 V=800.0 PL=0
MOVL C01699 V=800.0 PL=0
MOVL C01700 V=800.0 PL=0
MOVL C01701 V=800.0 PL=0
MOVL C01702 V=800.0 PL=0
MOVL C01703 V=800.0 PL=0
MOVL C01704 V=800.0 PL=0
MOVL C01705 V=800.0 PL=0
MOVL C01706 V=800.0 PL=0
MOVL C01707 V=800.0 PL=0
MOVL C01708 V=800.0 PL=0
MOVL C01709 V=800.0 PL=0
MOVL C01710 V=800.0 PL=0
MOVL C01711 V=800.0 PL=0
MOVL C01712 V=800.0 PL=0
MOVL C01713 V=800.0 PL=0
MOVL C01714 V=800.0 PL=0
MOVL C01715 V=800.0 PL=0
MOVL C01716 V=800.0 PL=0
MOVL C01717 V=800.0 PL=0
MOVL C01718 V=800.0 PL=0
MOVL C01719 V=800.0 PL=0
MOVL C01720 V=800.0 PL=0
MOVL C01721 V=800.0 PL=0
MOVL C01722 V=800.0 PL=0
MOVL C01723 V=800.0 PL=0
MOVL C01724 V=800.0 PL=0
MOVL C01725 V=800.0 PL=0
MOVL C01726 V=800.0 PL=0
MOVL C01727 V=800.0 PL=0
MOVL C01728 V=800.0 PL=0
MOVL C01729 V=800.0 PL=0
MOVL C01730 V=800.0 PL=0
MOVL C01731 V=800.0 PL=0
MOVL C01732 V=800.0 PL=0
MOVL C01733 V=800.0 PL=0
MOVL C01734 V=800.0 PL=0
MOVL C01735 V=800.0 PL=0
MOVL C01736 V=800.0 PL=0
MOVL C01737 V=800.0 PL=0
MOVL C01738 V=800.0 PL=0
MOVL C01739 V=800.0 PL=0
MOVL C01740 V=800.0 PL=0
MOVL C01741 V=800.0 PL=0
MOVL C01742 V=800.0 PL=0
MOVL C01743 V=800.0 PL=0
MOVL C01744 V=800.0 PL=0
MOVL C01745 V=800.0 PL=0
MOVL C01746 V=800.0 PL=0
MOVL C01747 V=800.0 PL=0
MOVL C01748 V=800.0 PL=0
MOVL C01749 V=800.0 PL=0
MOVL C01750 V=800.0 PL=0
MOVL C01751 V=800.0 PL=0
MOVL C01752 V=800.0 PL=0
MOVL C01753 V=800.0 PL=0
MOVL C01754 V=800.0 PL=0
MOVL C01755 V=800.0 PL=0
MOVL C01756 V=800.0 PL=0
MOVL C01757 V=800.0 PL=0
MOVL C01758 V=800.0 PL=0
MOVL C01759 V=800.0 PL=0
MOVL C01760 V=800.0 PL=0
MOVL C01761 V=800.0 PL=0
MOVL C01762 V=800.0 PL=0
MOVL C01763 V=800.0 PL=0
MOVL C01764 V=800.0 PL=0
MOVL C01765 V=800.0 PL=0
MOVL C01766 V=800.0 PL=0
MOVL C01767 V=800.0 PL=0
MOVL C01768 V=800.0 PL=0
MOVL C01769 V=800.0 PL=0
MOVL C01770 V=800.0 PL=0
MOVL C01771 V=800.0 PL=0
MOVL C01772 V=800.0 PL=0
MOVL C01773 V=800.0 PL=0
MOVL C01774 V=800.0 PL=0
MOVL C01775 V=800.0 PL=0
MOVL C01776 V=800.0 PL=0
MOVL C01777 V=800.0 PL=0
MOVL C01778 V=800.0 PL=0
MOVL C01779 V=800.0 PL=0
MOVL C01780 V=800.0 PL=0
MOVL C01781 V=800.0 PL=0
MOVL C01782 V=800.0 PL=0
MOVL C01783 V=800.0 PL=0
MOVL C01784 V=800.0 PL=0
MOVL C01785 V=800.0 PL=0
MOVL C01786 V=800.0 PL=0
MOVL C01787 V=800.0 PL=0
MOVL C01788 V=800.0 PL=0
MOVL C01789 V=800.0 PL=0
MOVL C01790 V=800.0 PL=0
MOVL C01791 V=800.0 PL=0
MOVL C01792 V=800.0 PL=0
MOVL C01793 V=800.0 PL=0
MOVL C01794 V=800.0 PL=0
MOVL C01795 V=800.0 PL=0
MOVL C01796 V=800.0 PL=0
MOVL C01797 V=800.0 PL=0
MOVL C01798 V=800.0 PL=0
MOVL C01799 V=800.0 PL=0
MOVL C01800 V=800.0 PL=0
MOVL C01801 V=800.0 PL=0
MOVL C01802 V=800.0 PL=0
MOVL C01803 V=800.0 PL=0
MOVL C01804 V=800.0 PL=0
MOVL C01805 V=800.0 PL=0
MOVL C01806 V=800.0 PL=0
MOVL C01807 V=800.0 PL=0
MOVL C01808 V=800.0 PL=0
MOVL C01809 V=800.0 PL=0
MOVL C01810 V=800.0 PL=0
MOVL C01811 V=800.0 PL=0
MOVL C01812 V=800.0 PL=0
MOVL C01813 V=800.0 PL=0
MOVL C01814 V=800.0 PL=0
MOVL C01815 V=800.0 PL=0
MOVL C01816 V=800.0 PL=0
MOVL C01817 V=800.0 PL=0
MOVL C01818 V=800.0 PL=0
MOVL C01819 V=800.0 PL=0
MOVL C01820 V=800.0 PL=0
MOVL C01821 V=800.0 PL=0
MOVL C01822 V=800.0 PL=0
MOVL C01823 V=800.0 PL=0
MOVL C01824 V=800.0 PL=0
MOVL C01825 V=800.0 PL=0
MOVL C01826 V=800.0 PL=0
MOVL C01827 V=800.0 PL=0
MOVL C01828 V=800.0 PL=0
MOVL C01829 V=800.0 PL=0
MOVL C01830 V=800.0 PL=0
MOVL C01831 V=800.0 PL=0
MOVL C01832 V=800.0 PL=0
MOVL C01833 V=800.0 PL=0
MOVL C01834 V=800.0 PL=0
MOVL C01835 V=800.0 PL=0
MOVL C01836 V=800.0 PL=0
MOVL C01837 V=800.0 PL=0
MOVL C01838 V=800.0 PL=0
MOVL C01839 V=800.0 PL=0
MOVL C01840 V=800.0 PL=0
MOVL C01841 V=800.0 PL=0
MOVL C01842 V=800.0 PL=0
MOVL C01843 V=800.0 PL=0
MOVL C01844 V=800.0 PL=0
MOVL C01845 V=800.0 PL=0
MOVL C01846 V=800.0 PL=0
MOVL C01847 V=800.0 PL=0
MOVL C01848 V=800.0 PL=0
MOVL C01849 V=800.0 PL=0
MOVL C01850 V=800.0 PL=0
MOVL C01851 V=800.0 PL=0
MOVL C01852 V=800.0 PL=0
MOVL C01853 V=800.0 PL=0
MOVL C01854 V=800.0 PL=0
MOVL C01855 V=800.0 PL=0
MOVL C01856 V=800.0 PL=0
MOVL C01857 V=800.0 PL=0
MOVL C01858 V=800.0 PL=0
MOVL C01859 V=800.0 PL=0
MOVL C01860 V=800.0 PL=0
MOVL C01861 V=800.0 PL=0
MOVL C01862 V=800.0 PL=0
MOVL C01863 V=800.0 PL=0
MOVL C01864 V=800.0 PL=0
MOVL C01865 V=800.0 PL=0
MOVL C01866 V=800.0 PL=0
MOVL C01867 V=800.0 PL=0
MOVL C01868 V=800.0 PL=0
MOVL C01869 V=800.0 PL=0
MOVL C01870 V=800.0 PL=0
MOVL C01871 V=800.0 PL=0
MOVL C01872 V=800.0 PL=0
MOVL C01873 V=800.0 PL=0
MOVL C01874 V=800.0 PL=0
MOVL C01875 V=800.0 PL=0
MOVL C01876 V=800.0 PL=0
MOVL C01877 V=800.0 PL=0
MOVL C01878 V=800.0 PL=0
MOVL C01879 V=800.0 PL=0
MOVL C01880 V=800.0 PL=0
MOVL C01881 V=800.0 PL=0
MOVL C01882 V=800.0 PL=0
MOVL C01883 V=800.0 PL=0
MOVL C01884 V=800.0 PL=0
MOVL C01885 V=800.0 PL=0
MOVL C01886 V=800.0 PL=0
MOVL C01887 V=800.0 PL=0
MOVL C01888 V=800.0 PL=0
MOVL C01889 V=800.0 PL=0
MOVL C01890 V=800.0 PL=0
MOVL C01891 V=800.0 PL=0
MOVL C01892 V=800.0 PL=0
MOVL C01893 V=800.0 PL=0
MOVL C01894 V=800.0 PL=0
MOVL C01895 V=800.0 PL=0
MOVL C01896 V=800.0 PL=0
MOVL C01897 V=800.0 PL=0
MOVL C01898 V=800.0 PL=0
MOVL C01899 V=800.0 PL=0
MOVL C01900 V=800.0 PL=0
MOVL C01901 V=800.0 PL=0
MOVL C01902 V=800.0 PL=0
MOVL C01903 V=800.0 PL=0
MOVL C01904 V=800.0 PL=0
MOVL C01905 V=800.0 PL=0
MOVL C01906 V=800.0 PL=0
MOVL C01907 V=800.0 PL=0
MOVL C01908 V=800.0 PL=0
MOVL C01909 V=800.0 PL=0
MOVL C01910 V=800.0 PL=0
MOVL C01911 V=800.0 PL=0
MOVL C01912 V=800.0 PL=0
MOVL C01913 V=800.0 PL=0
MOVL C01914 V=800.0 PL=0
MOVL C01915 V=800.0 PL=0
MOVL C01916 V=800.0 PL=0
MOVL C01917 V=800.0 PL=0
MOVL C01918 V=800.0 PL=0
MOVL C01919 V=800.0 PL=0
MOVL C01920 V=800.0 PL=0
MOVL C01921 V=800.0 PL=0
MOVL C01922 V=800.0 PL=0
MOVL C01923 V=800.0 PL=0
MOVL C01924 V=800.0 PL=0
MOVL C01925 V=800.0 PL=0
MOVL C01926 V=800.0 PL=0
MOVL C01927 V=800.0 PL=0
MOVL C01928 V=800.0 PL=0
MOVL C01929 V=800.0 PL=0
MOVL C01930 V=800.0 PL=0
MOVL C01931 V=800.0 PL=0
MOVL C01932 V=800.0 PL=0
MOVL C01933 V=800.0 PL=0
MOVL C01934 V=800.0 PL=0
MOVL C01935 V=800.0 PL=0
MOVL C01936 V=800.0 PL=0
MOVL C01937 V=800.0 PL=0
MOVL C01938 V=800.0 PL=0
MOVL C01939 V=800.0 PL=0
MOVL C01940 V=800.0 PL=0
MOVL C01941 V=800.0 PL=0
MOVL C01942 V=800.0 PL=0
MOVL C01943 V=800.0 PL=0
MOVL C01944 V=800.0 PL=0
MOVL C01945 V=800.0 PL=0
MOVL C01946 V=800.0 PL=0
MOVL C01947 V=800.0 PL=0
MOVL C01948 V=800.0 PL=0
MOVL C01949 V=800.0 PL=0
MOVL C01950 V=800.0 PL=0
MOVL C01951 V=800.0 PL=0
MOVL C01952 V=800.0 PL=0
MOVL C01953 V=800.0 PL=0
MOVL C01954 V=800.0 PL=0
MOVL C01955 V=800.0 PL=0
MOVL C01956 V=800.0 PL=0
MOVL C01957 V=800.0 PL=0
MOVL C01958 V=800.0 PL=0
MOVL C01959 V=800.0 PL=0
MOVL C01960 V=800.0 PL=0
MOVL C01961 V=800.0 PL=0
MOVL C01962 V=800.0 PL=0
MOVL C01963 V=800.0 PL=0
MOVL C01964 V=800.0 PL=0
MOVL C01965 V=800.0 PL=0
MOVL C01966 V=800.0 PL=0
MOVL C01967 V=800.0 PL=0
MOVL C01968 V=800.0 PL=0
MOVL C01969 V=800.0 PL=0
MOVL C01970 V=800.0 PL=0
MOVL C01971 V=800.0 PL=0
MOVL C01972 V=800.0 PL=0
MOVL C01973 V=800.0 PL=0
MOVL C01974 V=800.0 PL=0
MOVL C01975 V=800.0 PL=0
MOVL C01976 V=800.0 PL=0
MOVL C01977 V=800.0 PL=0
MOVL C01978 V=800.0 PL=0
MOVL C01979 V=800.0 PL=0
MOVL C01980 V=800.0 PL=0
MOVL C01981 V=800.0 PL=0
MOVL C01982 V=800.0 PL=0
MOVL C01983 V=800.0 PL=0
MOVL C01984 V=800.0 PL=0
MOVL C01985 V=800.0 PL=0
MOVL C01986 V=800.0 PL=0
MOVL C01987 V=800.0 PL=0
MOVL C01988 V=800.0 PL=0
MOVL C01989 V=800.0 PL=0
MOVL C01990 V=800.0 PL=0
MOVL C01991 V=800.0 PL=0
MOVL C01992 V=800.0 PL=0
MOVL C01993 V=800.0 PL=0
MOVL C01994 V=800.0 PL=0
MOVL C01995 V=800.0 PL=0
MOVL C01996 V=800.0 PL=0
MOVL C01997 V=800.0 PL=0
MOVL C01998 V=800.0 PL=0
MOVL C01999 V=800.0 PL=0
MOVL C02000 V=800.0 PL=0
MOVL C02001 V=800.0 PL=0
MOVL C02002 V=800.0 PL=0
MOVL C02003 V=800.0 PL=0
MOVL C02004 V=800.0 PL=0
MOVL C02005 V=800.0 PL=0
MOVL C02006 V=800.0 PL=0
MOVL C02007 V=800.0 PL=0
MOVL C02008 V=800.0 PL=0
MOVL C02009 V=800.0 PL=0
MOVL C02010 V=800.0 PL=0
MOVL C02011 V=800.0 PL=0
MOVL C02012 V=800.0 PL=0
MOVL C02013 V=800.0 PL=0
MOVL C02014 V=800.0 PL=0
MOVL C02015 V=800.0 PL=0
MOVL C02016 V=800.0 PL=0
MOVL C02017 V=800.0 PL=0
MOVL C02018 V=800.0 PL=0
MOVL C02019 V=800.0 PL=0
MOVL C02020 V=800.0 PL=0
MOVL C02021 V=800.0 PL=0
MOVL C02022 V=800.0 PL=0
MOVL C02023 V=800.0 PL=0
MOVL C02024 V=800.0 PL=0
MOVL C02025 V=800.0 PL=0
MOVL C02026 V=800.0 PL=0
MOVL C02027 V=800.0 PL=0
MOVL C02028 V=800.0 PL=0
MOVL C02029 V=800.0 PL=0
MOVL C02030 V=800.0 PL=0
MOVL C02031 V=800.0 PL=0
MOVL C02032 V=800.0 PL=0
MOVL C02033 V=800.0 PL=0
MOVL C02034 V=800.0 PL=0
MOVL C02035 V=800.0 PL=0
MOVL C02036 V=800.0 PL=0
MOVL C02037 V=800.0 PL=0
MOVL C02038 V=800.0 PL=0
